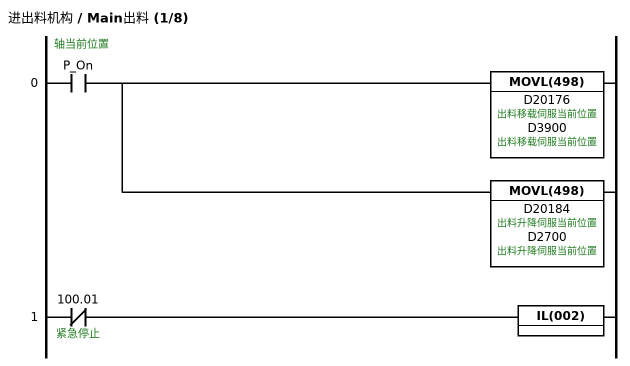
; [picture p48: 进出料机构 / Main出料, rungs 0-1]
; rung 0: 轴当前位置
LD P_On
MOVL(498) D20176 D3900  ; 出料移载伺服当前位置
MOVL(498) D20184 D2700  ; 出料升降伺服当前位置
; rung 1
LDNOT 100.01  ; 紧急停止
IL(002)

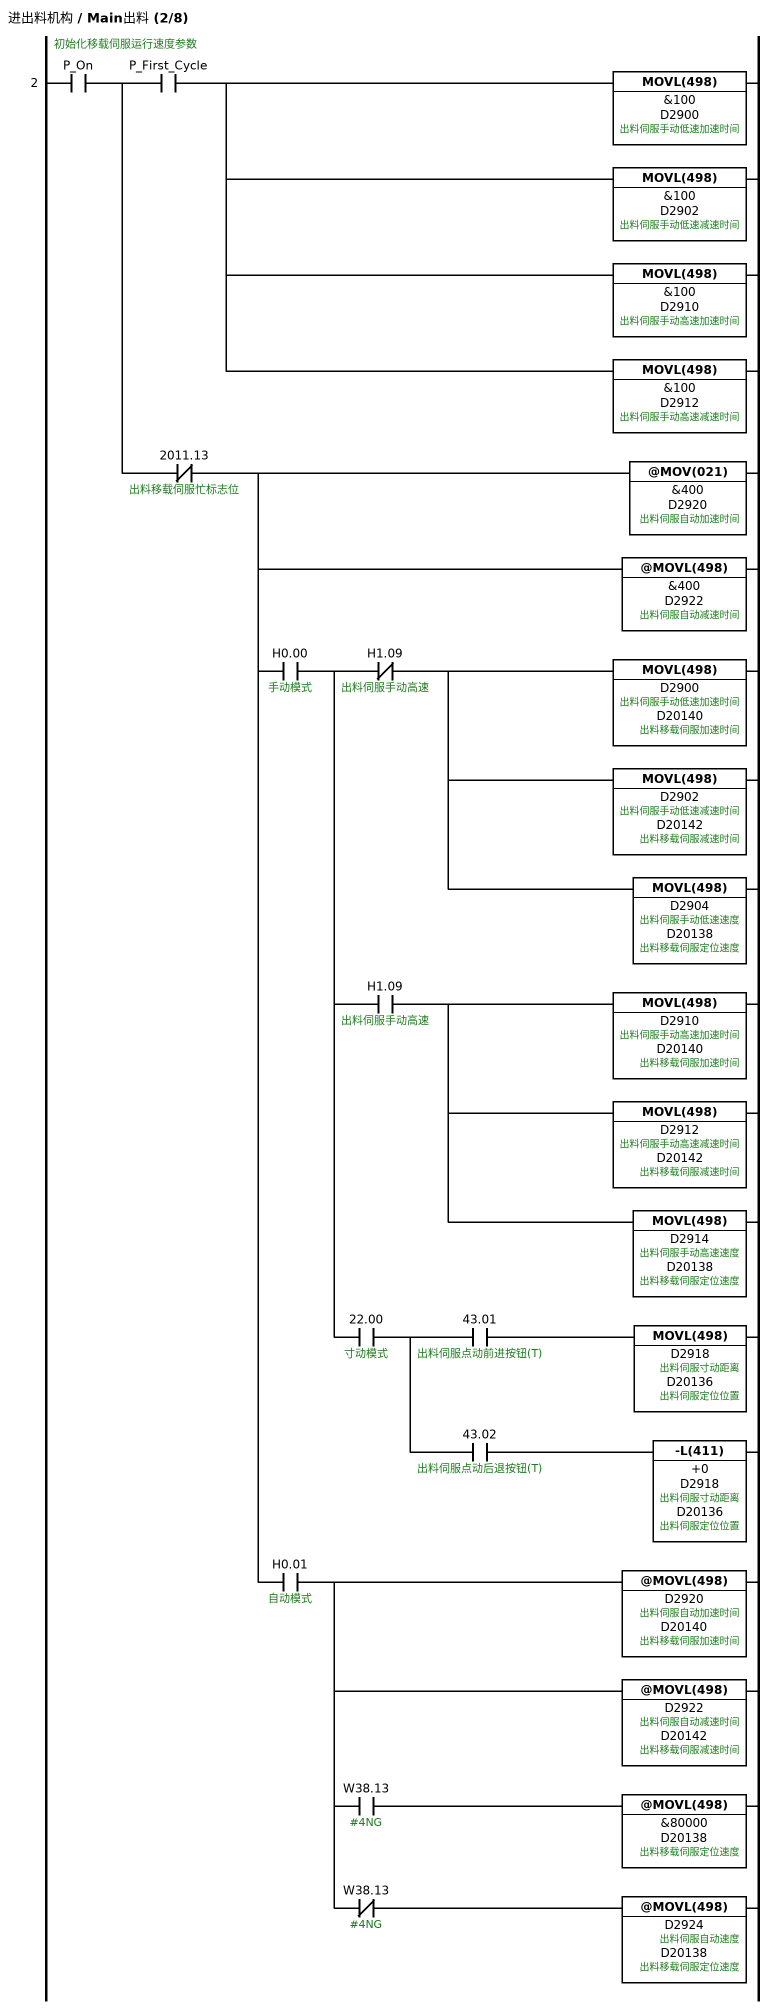
; rung 2: 初始化移载伺服运行速度参数
LD P_On
OUT TR0
AND P_First_Cycle
MOVL(498) &100 D2900  ; 出料伺服手动低速加速时间
MOVL(498) &100 D2902  ; 出料伺服手动低速减速时间
MOVL(498) &100 D2910  ; 出料伺服手动高速加速时间
MOVL(498) &100 D2912  ; 出料伺服手动高速减速时间
LD TR0
ANDNOT 2011.13  ; 出料移载伺服忙标志位
OUT TR0
@MOV(021) &400 D2920  ; 出料伺服自动加速时间
@MOVL(498) &400 D2922  ; 出料伺服自动减速时间
AND H0.00  ; 手动模式
OUT TR1
ANDNOT H1.09  ; 出料伺服手动高速
MOVL(498) D2900 D20140  ; 出料伺服手动低速加速时间, 出料移载伺服加速时间
MOVL(498) D2902 D20142  ; 出料伺服手动低速减速时间, 出料移载伺服减速时间
MOVL(498) D2904 D20138  ; 出料伺服手动低速速度, 出料移载伺服定位速度
LD TR1
AND H1.09  ; 出料伺服手动高速
MOVL(498) D2910 D20140  ; 出料伺服手动高速加速时间, 出料移载伺服加速时间
MOVL(498) D2912 D20142  ; 出料伺服手动高速减速时间, 出料移载伺服减速时间
MOVL(498) D2914 D20138  ; 出料伺服手动高速速度, 出料移载伺服定位速度
LD TR1
AND 22.00  ; 寸动模式
OUT TR1
AND 43.01  ; 出料伺服点动前进按钮(T)
MOVL(498) D2918 D20136  ; 出料伺服寸动距离, 出料伺服定位位置
LD TR1
AND 43.02  ; 出料伺服点动后退按钮(T)
-L(411) +0 D2918 D20136  ; 出料伺服寸动距离, 出料伺服定位位置
LD TR0
AND H0.01  ; 自动模式
OUT TR0
@MOVL(498) D2920 D20140  ; 出料伺服自动加速时间, 出料移载伺服加速时间
@MOVL(498) D2922 D20142  ; 出料伺服自动减速时间, 出料移载伺服减速时间
AND W38.13  ; #4NG
@MOVL(498) &80000 D20138  ; 出料移载伺服定位速度
LD TR0
ANDNOT W38.13  ; #4NG
@MOVL(498) D2924 D20138  ; 出料伺服自动速度, 出料移载伺服定位速度

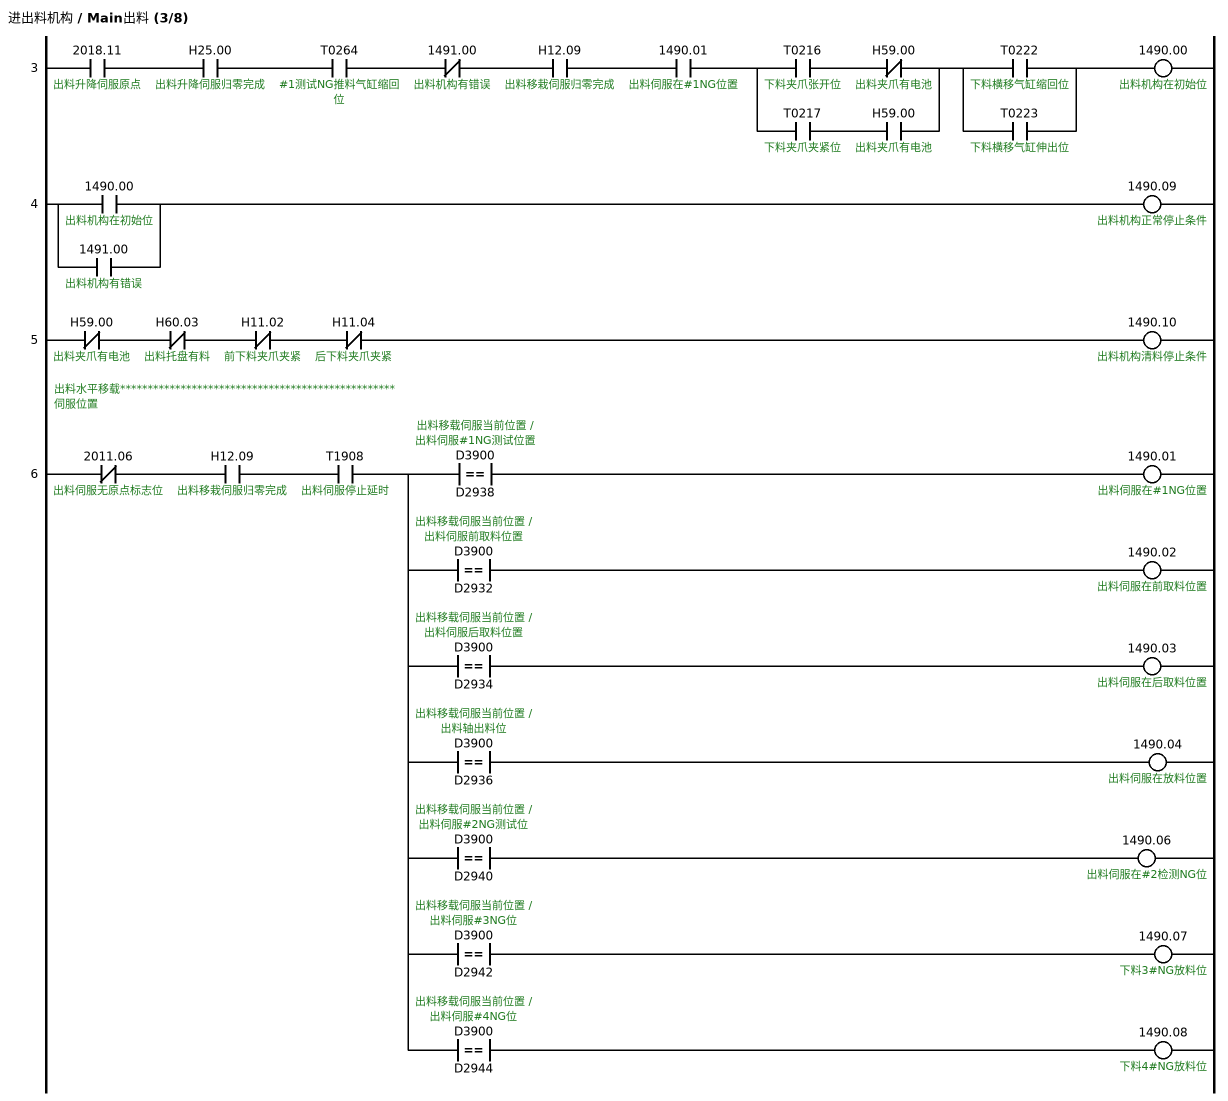
; rung 3
LD 2018.11  ; 出料升降伺服原点
AND H25.00  ; 出料升降伺服归零完成
AND T0264  ; #1测试NG推料气缸缩回位
ANDNOT 1491.00  ; 出料机构有错误
AND H12.09  ; 出料移栽伺服归零完成
AND 1490.01  ; 出料伺服在#1NG位置
LD T0216  ; 下料夹爪张开位
ANDNOT H59.00  ; 出料夹爪有电池
LD T0217  ; 下料夹爪夹紧位
AND H59.00  ; 出料夹爪有电池
ORLD
ANDLD
LD T0222  ; 下料横移气缸缩回位
OR T0223  ; 下料横移气缸伸出位
ANDLD
OUT 1490.00  ; 出料机构在初始位
; rung 4
LD 1490.00  ; 出料机构在初始位
OR 1491.00  ; 出料机构有错误
OUT 1490.09  ; 出料机构正常停止条件
; rung 5
LDNOT H59.00  ; 出料夹爪有电池
ANDNOT H60.03  ; 出料托盘有料
ANDNOT H11.02  ; 前下料夹爪夹紧
ANDNOT H11.04  ; 后下料夹爪夹紧
OUT 1490.10  ; 出料机构清料停止条件
; rung 6: 出料水平移载************************************************** / 伺服位置
LDNOT 2011.06  ; 出料伺服无原点标志位
AND H12.09  ; 出料移栽伺服归零完成
AND T1908  ; 出料伺服停止延时
OUT TR0
AND=SL(303) D3900 D2938  ; 出料移载伺服当前位置, 出料伺服#1NG测试位置
OUT 1490.01  ; 出料伺服在#1NG位置
LD TR0
AND=SL(303) D3900 D2932  ; 出料移载伺服当前位置, 出料伺服前取料位置
OUT 1490.02  ; 出料伺服在前取料位置
LD TR0
AND=SL(303) D3900 D2934  ; 出料移载伺服当前位置, 出料伺服后取料位置
OUT 1490.03  ; 出料伺服在后取料位置
LD TR0
AND=SL(303) D3900 D2936  ; 出料移载伺服当前位置, 出料轴出料位
OUT 1490.04  ; 出料伺服在放料位置
LD TR0
AND=SL(303) D3900 D2940  ; 出料移载伺服当前位置, 出料伺服#2NG测试位
OUT 1490.06  ; 出料伺服在#2检测NG位
LD TR0
AND=SL(303) D3900 D2942  ; 出料移载伺服当前位置, 出料伺服#3NG位
OUT 1490.07  ; 下料3#NG放料位
LD TR0
AND=SL(303) D3900 D2944  ; 出料移载伺服当前位置, 出料伺服#4NG位
OUT 1490.08  ; 下料4#NG放料位

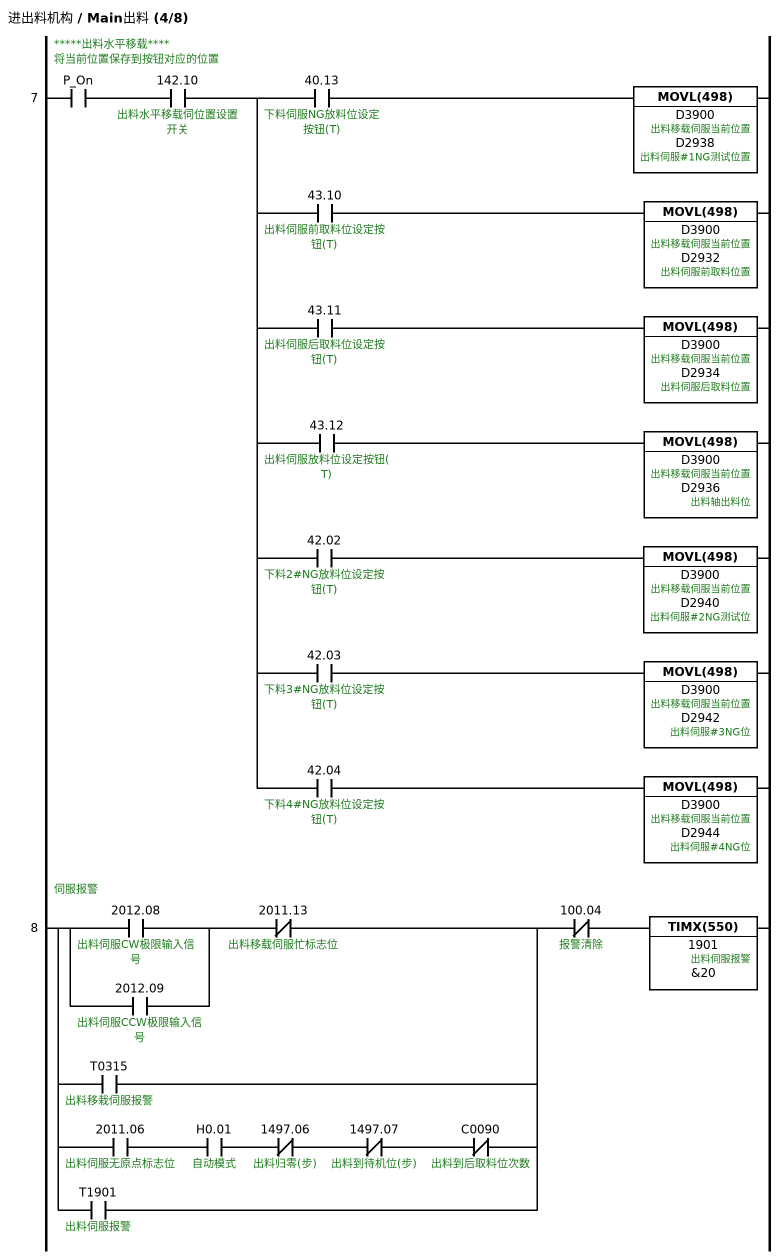
; rung 7: *****出料水平移载**** / 将当前位置保存到按钮对应的位置
LD P_On
AND 142.10  ; 出料水平移载伺位置设置开关
OUT TR0
AND 40.13  ; 下料伺服NG放料位设定按钮(T)
MOVL(498) D3900 D2938  ; 出料移载伺服当前位置, 出料伺服#1NG测试位置
LD TR0
AND 43.10  ; 出料伺服前取料位设定按钮(T)
MOVL(498) D3900 D2932  ; 出料移载伺服当前位置, 出料伺服前取料位置
LD TR0
AND 43.11  ; 出料伺服后取料位设定按钮(T)
MOVL(498) D3900 D2934  ; 出料移载伺服当前位置, 出料伺服后取料位置
LD TR0
AND 43.12  ; 出料伺服放料位设定按钮(T)
MOVL(498) D3900 D2936  ; 出料移载伺服当前位置, 出料轴出料位
LD TR0
AND 42.02  ; 下料2#NG放料位设定按钮(T)
MOVL(498) D3900 D2940  ; 出料移载伺服当前位置, 出料伺服#2NG测试位
LD TR0
AND 42.03  ; 下料3#NG放料位设定按钮(T)
MOVL(498) D3900 D2942  ; 出料移载伺服当前位置, 出料伺服#3NG位
LD TR0
AND 42.04  ; 下料4#NG放料位设定按钮(T)
MOVL(498) D3900 D2944  ; 出料移载伺服当前位置, 出料伺服#4NG位
; rung 8: 伺服报警
LD 2012.08  ; 出料伺服CW极限输入信号
OR 2012.09  ; 出料伺服CCW极限输入信号
ANDNOT 2011.13  ; 出料移载伺服忙标志位
OR T0315  ; 出料移栽伺服报警
LD 2011.06  ; 出料伺服无原点标志位
AND H0.01  ; 自动模式
ANDNOT 1497.06  ; 出料归零(步)
ANDNOT 1497.07  ; 出料到待机位(步)
ANDNOT C0090  ; 出料到后取料位次数
ORLD
OR T1901  ; 出料伺服报警
ANDNOT 100.04  ; 报警清除
TIMX(550) 1901 &20  ; 出料伺服报警

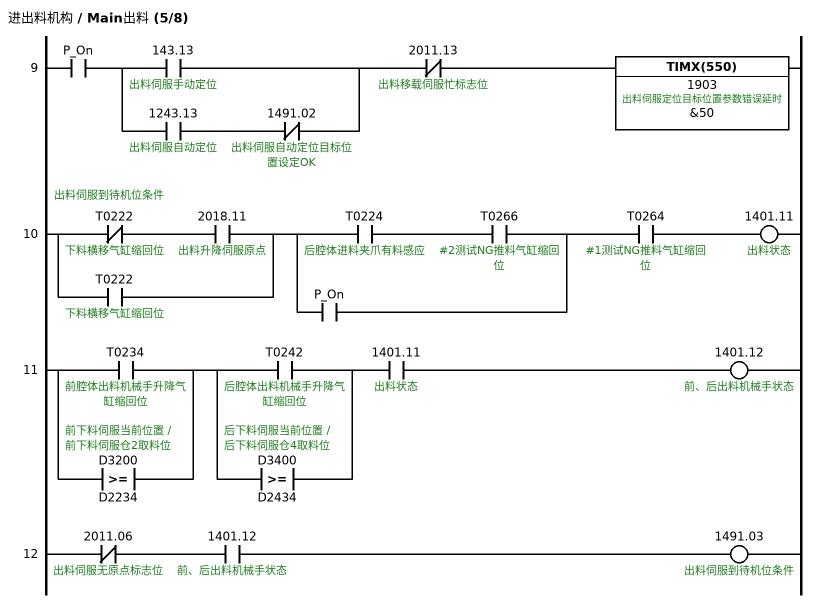
; rung 9
LD P_On
LD 143.13  ; 出料伺服手动定位
LD 1243.13  ; 出料伺服自动定位
ANDNOT 1491.02  ; 出料伺服自动定位目标位置设定OK
ORLD
ANDLD
ANDNOT 2011.13  ; 出料移载伺服忙标志位
TIMX(550) 1903 &50  ; 出料伺服定位目标位置参数错误延时
; rung 10: 出料伺服到待机位条件
LDNOT T0222  ; 下料横移气缸缩回位
AND 2018.11  ; 出料升降伺服原点
OR T0222  ; 下料横移气缸缩回位
LD T0224  ; 后腔体进料夹爪有料感应
AND T0266  ; #2测试NG推料气缸缩回位
OR P_On
ANDLD
AND T0264  ; #1测试NG推料气缸缩回位
OUT 1401.11  ; 出料状态
; rung 11
LD T0234  ; 前腔体出料机械手升降气缸缩回位
OR>=SL(328) D3200 D2234  ; 前下料伺服当前位置, 前下料伺服仓2取料位
LD T0242  ; 后腔体出料机械手升降气缸缩回位
OR>=SL(328) D3400 D2434  ; 后下料伺服当前位置, 后下料伺服仓4取料位
ANDLD
AND 1401.11  ; 出料状态
OUT 1401.12  ; 前、后出料机械手状态
; rung 12
LDNOT 2011.06  ; 出料伺服无原点标志位
AND 1401.12  ; 前、后出料机械手状态
OUT 1491.03  ; 出料伺服到待机位条件

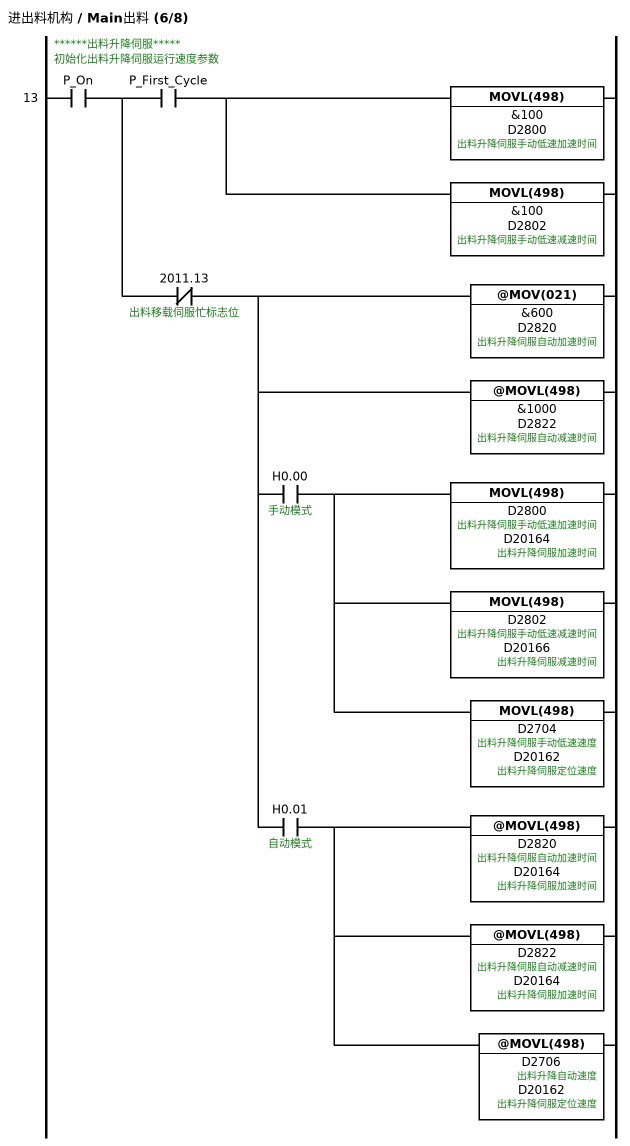
; rung 13: ******出料升降伺服***** / 初始化出料升降伺服运行速度参数
LD P_On
OUT TR0
AND P_First_Cycle
MOVL(498) &100 D2800  ; 出料升降伺服手动低速加速时间
MOVL(498) &100 D2802  ; 出料升降伺服手动低速减速时间
LD TR0
ANDNOT 2011.13  ; 出料移载伺服忙标志位
OUT TR0
@MOV(021) &600 D2820  ; 出料升降伺服自动加速时间
@MOVL(498) &1000 D2822  ; 出料升降伺服自动减速时间
AND H0.00  ; 手动模式
MOVL(498) D2800 D20164  ; 出料升降伺服手动低速加速时间, 出料升降伺服加速时间
MOVL(498) D2802 D20166  ; 出料升降伺服手动低速减速时间, 出料升降伺服减速时间
MOVL(498) D2704 D20162  ; 出料升降伺服手动低速速度, 出料升降伺服定位速度
LD TR0
AND H0.01  ; 自动模式
@MOVL(498) D2820 D20164  ; 出料升降伺服自动加速时间, 出料升降伺服加速时间
@MOVL(498) D2822 D20164  ; 出料升降伺服自动减速时间, 出料升降伺服加速时间
@MOVL(498) D2706 D20162  ; 出料升降自动速度, 出料升降伺服定位速度

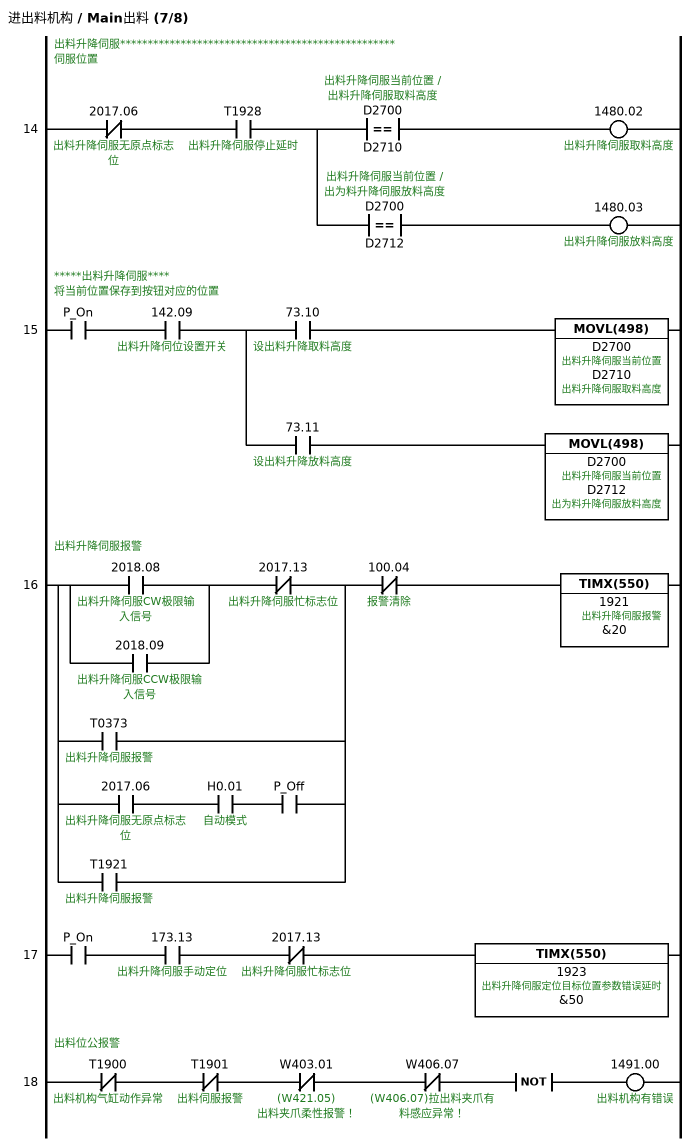
; rung 14: 出料升降伺服************************************************** / 伺服位置
LDNOT 2017.06  ; 出料升降伺服无原点标志位
AND T1928  ; 出料升降伺服停止延时
OUT TR0
AND=SL(303) D2700 D2710  ; 出料升降伺服当前位置, 出料升降伺服取料高度
OUT 1480.02  ; 出料升降伺服取料高度
LD TR0
AND=SL(303) D2700 D2712  ; 出料升降伺服当前位置, 出为料升降伺服放料高度
OUT 1480.03  ; 出料升降伺服放料高度
; rung 15: *****出料升降伺服**** / 将当前位置保存到按钮对应的位置
LD P_On
AND 142.09  ; 出料升降伺位设置开关
OUT TR0
AND 73.10  ; 设出料升降取料高度
MOVL(498) D2700 D2710  ; 出料升降伺服当前位置, 出料升降伺服取料高度
LD TR0
AND 73.11  ; 设出料升降放料高度
MOVL(498) D2700 D2712  ; 出料升降伺服当前位置, 出为料升降伺服放料高度
; rung 16: 出料升降伺服报警
LD 2018.08  ; 出料升降伺服CW极限输入信号
OR 2018.09  ; 出料升降伺服CCW极限输入信号
ANDNOT 2017.13  ; 出料升降伺服忙标志位
OR T0373  ; 出料升降伺服报警
LD 2017.06  ; 出料升降伺服无原点标志位
AND H0.01  ; 自动模式
AND P_Off
ORLD
OR T1921  ; 出料升降伺服报警
ANDNOT 100.04  ; 报警清除
TIMX(550) 1921 &20  ; 出料升降伺服报警
; rung 17
LD P_On
AND 173.13  ; 出料升降伺服手动定位
ANDNOT 2017.13  ; 出料升降伺服忙标志位
TIMX(550) 1923 &50  ; 出料升降伺服定位目标位置参数错误延时
; rung 18: 出料位公报警
LDNOT T1900  ; 出料机构气缸动作异常
ANDNOT T1901  ; 出料伺服报警
ANDNOT W403.01  ; (W421.05) 出料夹爪柔性报警！
ANDNOT W406.07  ; (W406.07)拉出料夹爪有料感应异常！
NOT(520)
OUT 1491.00  ; 出料机构有错误

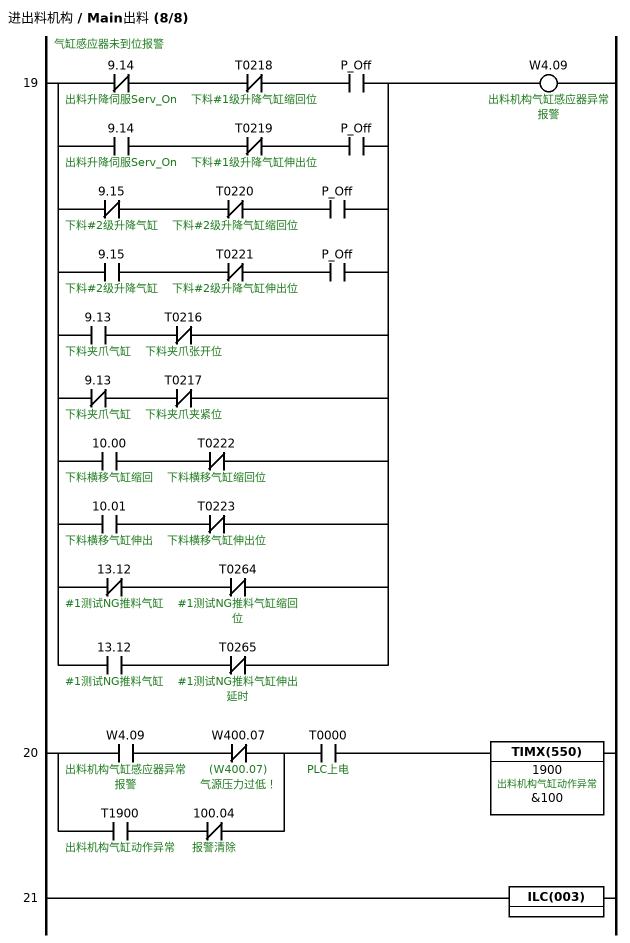
; rung 19: 气缸感应器未到位报警
LDNOT 9.14  ; 出料升降伺服Serv_On
ANDNOT T0218  ; 下料#1级升降气缸缩回位
AND P_Off
LD 9.14  ; 出料升降伺服Serv_On
ANDNOT T0219  ; 下料#1级升降气缸伸出位
AND P_Off
ORLD
LDNOT 9.15  ; 下料#2级升降气缸
ANDNOT T0220  ; 下料#2级升降气缸缩回位
AND P_Off
ORLD
LD 9.15  ; 下料#2级升降气缸
ANDNOT T0221  ; 下料#2级升降气缸伸出位
AND P_Off
ORLD
LD 9.13  ; 下料夹爪气缸
ANDNOT T0216  ; 下料夹爪张开位
ORLD
LDNOT 9.13  ; 下料夹爪气缸
ANDNOT T0217  ; 下料夹爪夹紧位
ORLD
LD 10.00  ; 下料横移气缸缩回
ANDNOT T0222  ; 下料横移气缸缩回位
ORLD
LD 10.01  ; 下料横移气缸伸出
ANDNOT T0223  ; 下料横移气缸伸出位
ORLD
LDNOT 13.12  ; #1测试NG推料气缸
ANDNOT T0264  ; #1测试NG推料气缸缩回位
ORLD
LD 13.12  ; #1测试NG推料气缸
ANDNOT T0265  ; #1测试NG推料气缸伸出延时
ORLD
OUT W4.09  ; 出料机构气缸感应器异常报警
; rung 20
LD W4.09  ; 出料机构气缸感应器异常报警
ANDNOT W400.07  ; (W400.07) 气源压力过低！
LD T1900  ; 出料机构气缸动作异常
ANDNOT 100.04  ; 报警清除
ORLD
AND T0000  ; PLC上电
TIMX(550) 1900 &100  ; 出料机构气缸动作异常
; rung 21
ILC(003)

### Section 工站复位

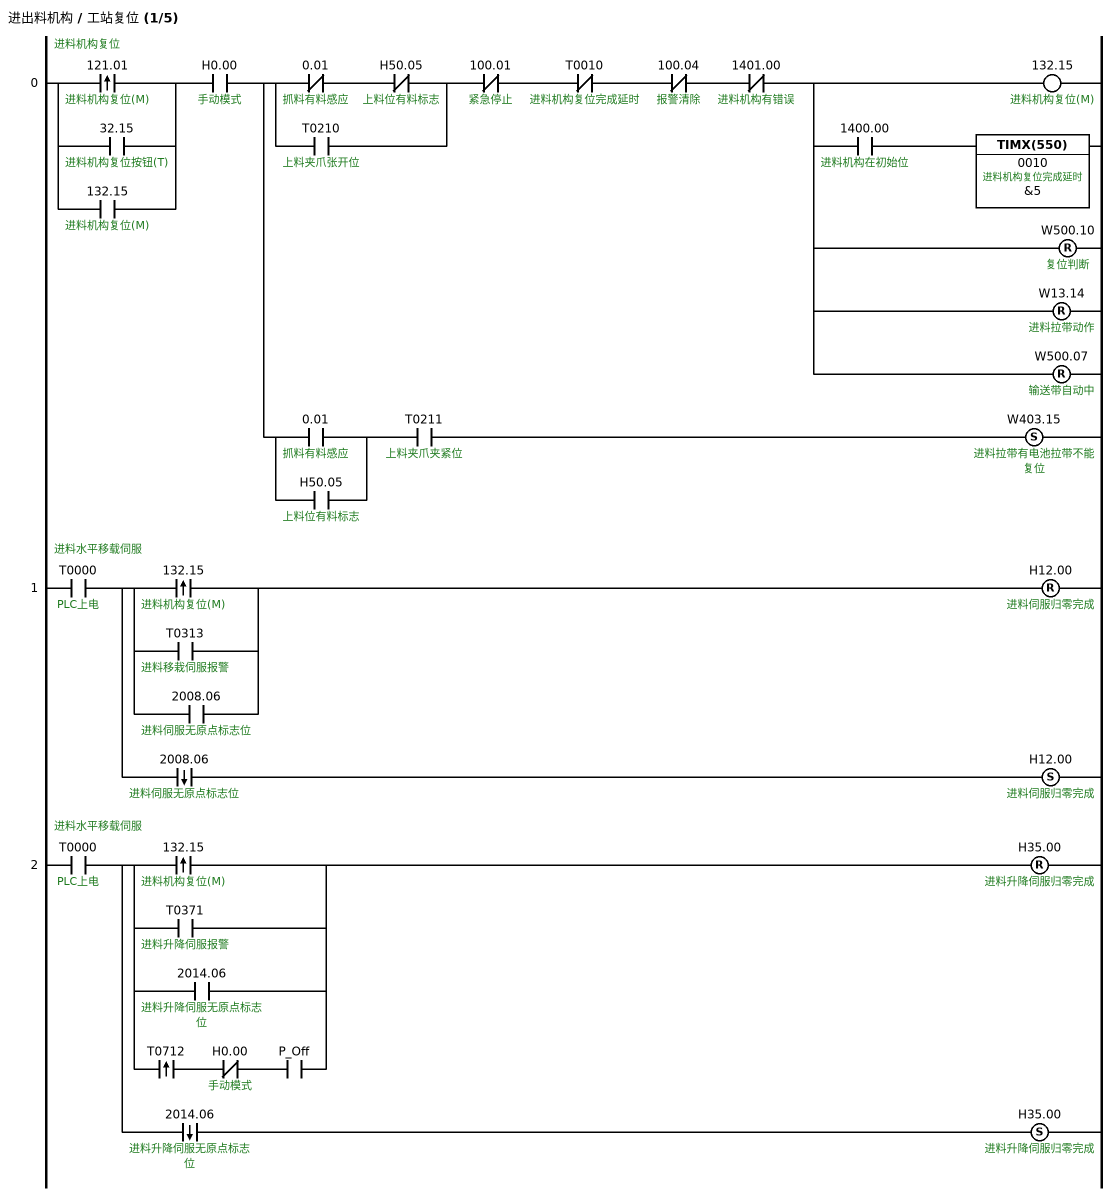
; rung 0: 进料机构复位
@LD 121.01  ; 进料机构复位(M)
OR 32.15  ; 进料机构复位按钮(T)
OR 132.15  ; 进料机构复位(M)
AND H0.00  ; 手动模式
OUT TR0
LDNOT 0.01  ; 抓料有料感应
ANDNOT H50.05  ; 上料位有料标志
OR T0210  ; 上料夹爪张开位
ANDLD
ANDNOT 100.01  ; 紧急停止
ANDNOT T0010  ; 进料机构复位完成延时
ANDNOT 100.04  ; 报警清除
ANDNOT 1401.00  ; 进料机构有错误
OUT TR1
OUT 132.15  ; 进料机构复位(M)
AND 1400.00  ; 进料机构在初始位
TIMX(550) 0010 &5  ; 进料机构复位完成延时
LD TR1
RSET W500.10  ; 复位判断
RSET W13.14  ; 进料拉带动作
RSET W500.07  ; 输送带自动中
LD TR0
LD 0.01  ; 抓料有料感应
OR H50.05  ; 上料位有料标志
ANDLD
AND T0211  ; 上料夹爪夹紧位
SET W403.15  ; 进料拉带有电池拉带不能复位
; rung 1: 进料水平移载伺服
LD T0000  ; PLC上电
OUT TR0
@LD 132.15  ; 进料机构复位(M)
OR T0313  ; 进料移栽伺服报警
OR 2008.06  ; 进料伺服无原点标志位
ANDLD
RSET H12.00  ; 进料伺服归零完成
LD TR0
%AND 2008.06  ; 进料伺服无原点标志位
SET H12.00  ; 进料伺服归零完成
; rung 2: 进料水平移载伺服
LD T0000  ; PLC上电
OUT TR0
@LD 132.15  ; 进料机构复位(M)
OR T0371  ; 进料升降伺服报警
OR 2014.06  ; 进料升降伺服无原点标志位
@LD T0712
ANDNOT H0.00  ; 手动模式
AND P_Off
ORLD
ANDLD
RSET H35.00  ; 进料升降伺服归零完成
LD TR0
%AND 2014.06  ; 进料升降伺服无原点标志位
SET H35.00  ; 进料升降伺服归零完成

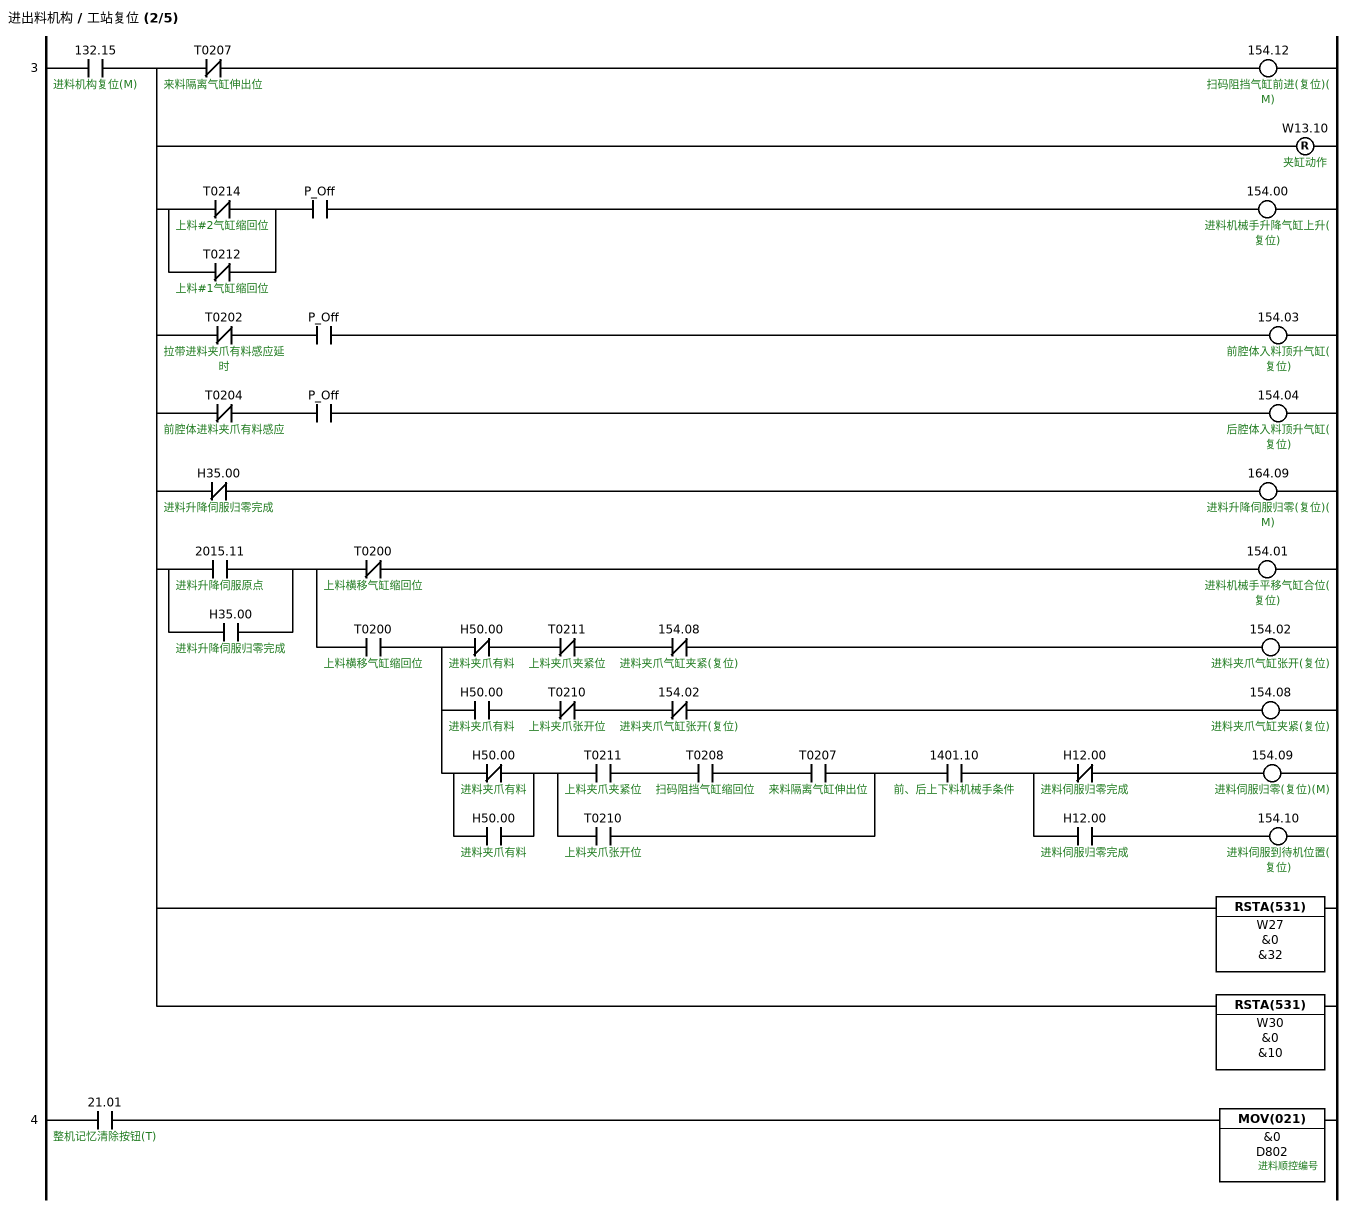
; rung 3
LD 132.15  ; 进料机构复位(M)
OUT TR0
ANDNOT T0207  ; 来料隔离气缸伸出位
OUT 154.12  ; 扫码阻挡气缸前进(复位)(M)
LD TR0
RSET W13.10  ; 夹缸动作
LDNOT T0214  ; 上料#2气缸缩回位
ORNOT T0212  ; 上料#1气缸缩回位
ANDLD
AND P_Off
OUT 154.00  ; 进料机械手升降气缸上升(复位)
LD TR0
ANDNOT T0202  ; 拉带进料夹爪有料感应延时
AND P_Off
OUT 154.03  ; 前腔体入料顶升气缸(复位)
LD TR0
ANDNOT T0204  ; 前腔体进料夹爪有料感应
AND P_Off
OUT 154.04  ; 后腔体入料顶升气缸(复位)
LD TR0
ANDNOT H35.00  ; 进料升降伺服归零完成
OUT 164.09  ; 进料升降伺服归零(复位)(M)
LD TR0
LD 2015.11  ; 进料升降伺服原点
OR H35.00  ; 进料升降伺服归零完成
ANDLD
OUT TR1
ANDNOT T0200  ; 上料横移气缸缩回位
OUT 154.01  ; 进料机械手平移气缸合位(复位)
LD TR1
AND T0200  ; 上料横移气缸缩回位
OUT TR1
ANDNOT H50.00  ; 进料夹爪有料
ANDNOT T0211  ; 上料夹爪夹紧位
ANDNOT 154.08  ; 进料夹爪气缸夹紧(复位)
OUT 154.02  ; 进料夹爪气缸张开(复位)
LD TR1
AND H50.00  ; 进料夹爪有料
ANDNOT T0210  ; 上料夹爪张开位
ANDNOT 154.02  ; 进料夹爪气缸张开(复位)
OUT 154.08  ; 进料夹爪气缸夹紧(复位)
LD TR1
LDNOT H50.00  ; 进料夹爪有料
OR H50.00  ; 进料夹爪有料
ANDLD
LD T0211  ; 上料夹爪夹紧位
AND T0208  ; 扫码阻挡气缸缩回位
AND T0207  ; 来料隔离气缸伸出位
OR T0210  ; 上料夹爪张开位
ANDLD
AND 1401.10  ; 前、后上下料机械手条件
OUT TR1
ANDNOT H12.00  ; 进料伺服归零完成
OUT 154.09  ; 进料伺服归零(复位)(M)
LD TR1
AND H12.00  ; 进料伺服归零完成
OUT 154.10  ; 进料伺服到待机位置(复位)
LD TR0
RSTA(531) W27 &0 &32
RSTA(531) W30 &0 &10
; rung 4
LD 21.01  ; 整机记忆清除按钮(T)
MOV(021) &0 D802  ; 进料顺控编号

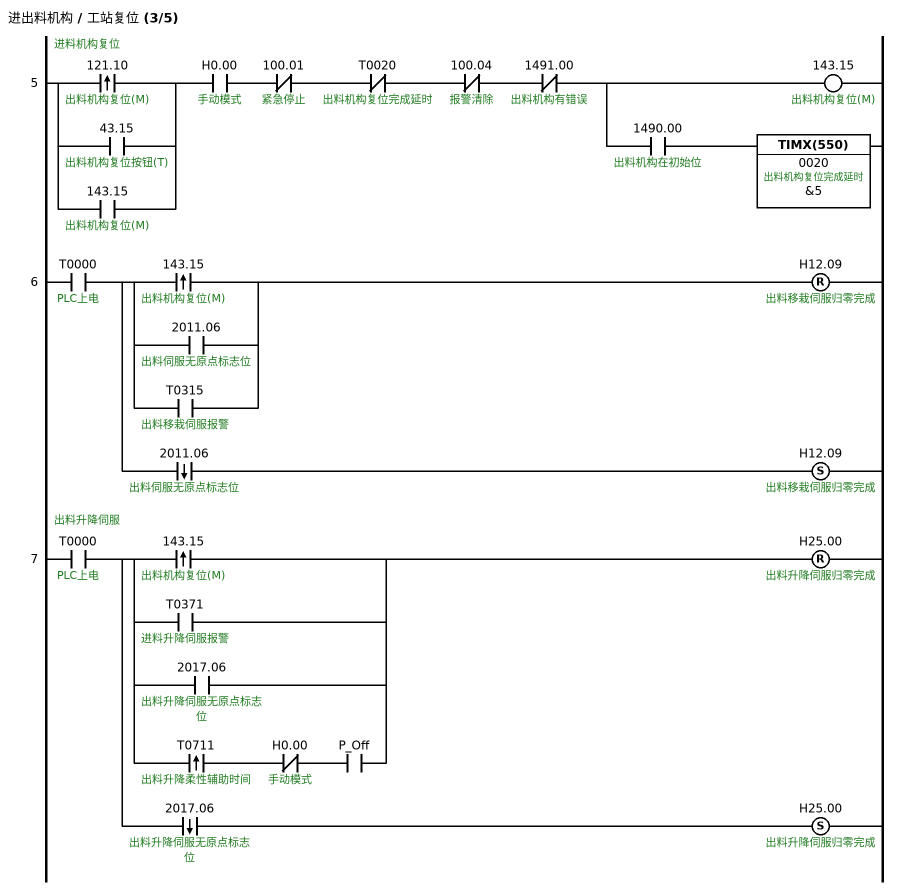
; rung 5: 进料机构复位
@LD 121.10  ; 出料机构复位(M)
OR 43.15  ; 出料机构复位按钮(T)
OR 143.15  ; 出料机构复位(M)
AND H0.00  ; 手动模式
ANDNOT 100.01  ; 紧急停止
ANDNOT T0020  ; 出料机构复位完成延时
ANDNOT 100.04  ; 报警清除
ANDNOT 1491.00  ; 出料机构有错误
OUT 143.15  ; 出料机构复位(M)
AND 1490.00  ; 出料机构在初始位
TIMX(550) 0020 &5  ; 出料机构复位完成延时
; rung 6
LD T0000  ; PLC上电
OUT TR0
@LD 143.15  ; 出料机构复位(M)
OR 2011.06  ; 出料伺服无原点标志位
OR T0315  ; 出料移栽伺服报警
ANDLD
RSET H12.09  ; 出料移栽伺服归零完成
LD TR0
%AND 2011.06  ; 出料伺服无原点标志位
SET H12.09  ; 出料移栽伺服归零完成
; rung 7: 出料升降伺服
LD T0000  ; PLC上电
OUT TR0
@LD 143.15  ; 出料机构复位(M)
OR T0371  ; 进料升降伺服报警
OR 2017.06  ; 出料升降伺服无原点标志位
@LD T0711  ; 出料升降柔性辅助时间
ANDNOT H0.00  ; 手动模式
AND P_Off
ORLD
ANDLD
RSET H25.00  ; 出料升降伺服归零完成
LD TR0
%AND 2017.06  ; 出料升降伺服无原点标志位
SET H25.00  ; 出料升降伺服归零完成

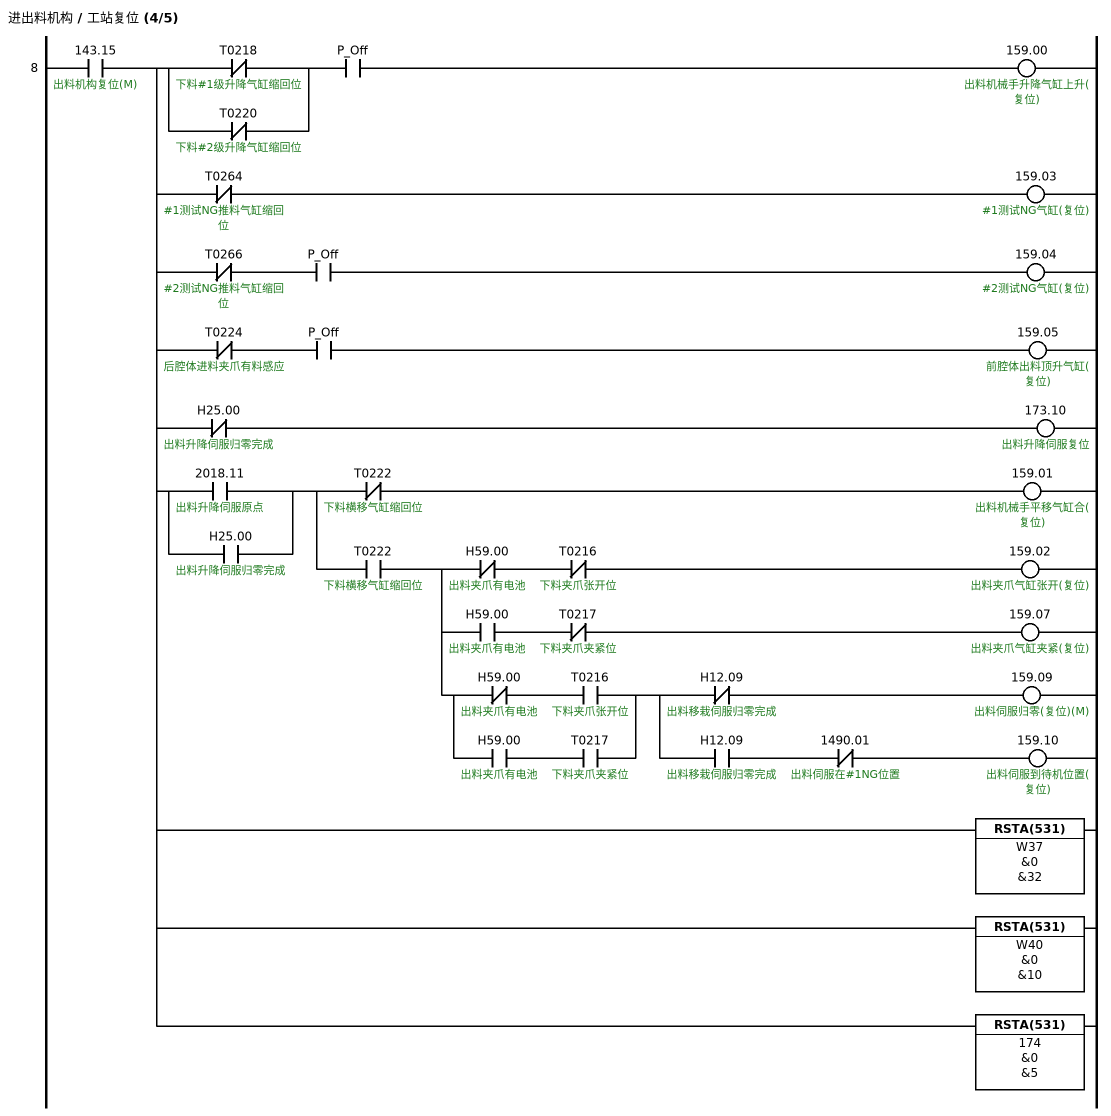
; rung 8
LD 143.15  ; 出料机构复位(M)
OUT TR0
LDNOT T0218  ; 下料#1级升降气缸缩回位
ORNOT T0220  ; 下料#2级升降气缸缩回位
ANDLD
AND P_Off
OUT 159.00  ; 出料机械手升降气缸上升(复位)
LD TR0
ANDNOT T0264  ; #1测试NG推料气缸缩回位
OUT 159.03  ; #1测试NG气缸(复位)
LD TR0
ANDNOT T0266  ; #2测试NG推料气缸缩回位
AND P_Off
OUT 159.04  ; #2测试NG气缸(复位)
LD TR0
ANDNOT T0224  ; 后腔体进料夹爪有料感应
AND P_Off
OUT 159.05  ; 前腔体出料顶升气缸(复位)
LD TR0
ANDNOT H25.00  ; 出料升降伺服归零完成
OUT 173.10  ; 出料升降伺服复位
LD TR0
LD 2018.11  ; 出料升降伺服原点
OR H25.00  ; 出料升降伺服归零完成
ANDLD
OUT TR1
ANDNOT T0222  ; 下料横移气缸缩回位
OUT 159.01  ; 出料机械手平移气缸合(复位)
LD TR1
AND T0222  ; 下料横移气缸缩回位
OUT TR1
ANDNOT H59.00  ; 出料夹爪有电池
ANDNOT T0216  ; 下料夹爪张开位
OUT 159.02  ; 出料夹爪气缸张开(复位)
LD TR1
AND H59.00  ; 出料夹爪有电池
ANDNOT T0217  ; 下料夹爪夹紧位
OUT 159.07  ; 出料夹爪气缸夹紧(复位)
LD TR1
LDNOT H59.00  ; 出料夹爪有电池
AND T0216  ; 下料夹爪张开位
LD H59.00  ; 出料夹爪有电池
AND T0217  ; 下料夹爪夹紧位
ORLD
ANDLD
OUT TR1
ANDNOT H12.09  ; 出料移栽伺服归零完成
OUT 159.09  ; 出料伺服归零(复位)(M)
LD TR1
AND H12.09  ; 出料移栽伺服归零完成
ANDNOT 1490.01  ; 出料伺服在#1NG位置
OUT 159.10  ; 出料伺服到待机位置(复位)
LD TR0
RSTA(531) W37 &0 &32
RSTA(531) W40 &0 &10
RSTA(531) 174 &0 &5

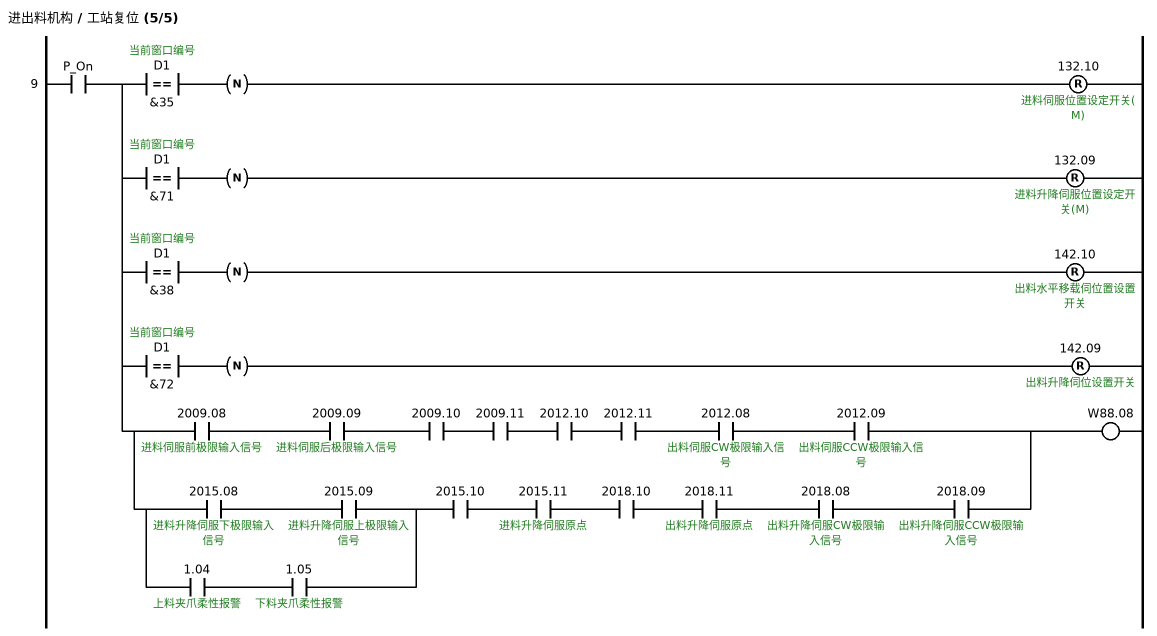
; rung 9
LD P_On
OUT TR0
AND=(300) D1 &35  ; 当前窗口编号
DOWN(522)
RSET 132.10  ; 进料伺服位置设定开关(M)
LD TR0
AND=(300) D1 &71  ; 当前窗口编号
DOWN(522)
RSET 132.09  ; 进料升降伺服位置设定开关(M)
LD TR0
AND=(300) D1 &38  ; 当前窗口编号
DOWN(522)
RSET 142.10  ; 出料水平移载伺位置设置开关
LD TR0
AND=(300) D1 &72  ; 当前窗口编号
DOWN(522)
RSET 142.09  ; 出料升降伺位设置开关
LD TR0
LD 2009.08  ; 进料伺服前极限输入信号
AND 2009.09  ; 进料伺服后极限输入信号
AND 2009.10
AND 2009.11
AND 2012.10
AND 2012.11
AND 2012.08  ; 出料伺服CW极限输入信号
AND 2012.09  ; 出料伺服CCW极限输入信号
LD 2015.08  ; 进料升降伺服下极限输入信号
AND 2015.09  ; 进料升降伺服上极限输入信号
LD 1.04  ; 上料夹爪柔性报警
AND 1.05  ; 下料夹爪柔性报警
ORLD
AND 2015.10
AND 2015.11  ; 进料升降伺服原点
AND 2018.10
AND 2018.11  ; 出料升降伺服原点
AND 2018.08  ; 出料升降伺服CW极限输入信号
AND 2018.09  ; 出料升降伺服CCW极限输入信号
ORLD
ANDLD
OUT W88.08

### Section 扫码

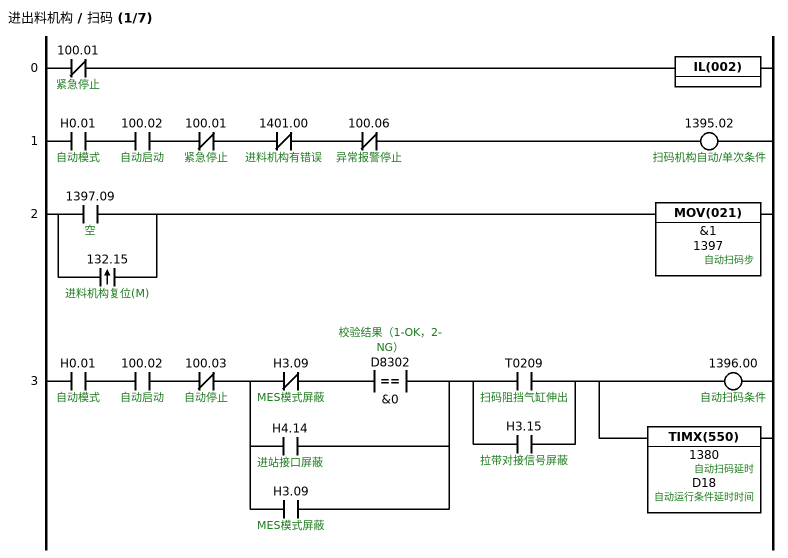
; rung 0
LDNOT 100.01  ; 紧急停止
IL(002)
; rung 1
LD H0.01  ; 自动模式
AND 100.02  ; 自动启动
ANDNOT 100.01  ; 紧急停止
ANDNOT 1401.00  ; 进料机构有错误
ANDNOT 100.06  ; 异常报警停止
OUT 1395.02  ; 扫码机构自动/单次条件
; rung 2
LD 1397.09  ; 空
@OR 132.15  ; 进料机构复位(M)
MOV(021) &1 1397  ; 自动扫码步
; rung 3
LD H0.01  ; 自动模式
AND 100.02  ; 自动启动
ANDNOT 100.03  ; 自动停止
LDNOT H3.09  ; MES模式屏蔽
AND=(300) D8302 &0  ; 校验结果（1-OK，2-NG）
OR H4.14  ; 进站接口屏蔽
OR H3.09  ; MES模式屏蔽
ANDLD
LD T0209  ; 扫码阻挡气缸伸出
OR H3.15  ; 拉带对接信号屏蔽
ANDLD
OUT 1396.00  ; 自动扫码条件
TIMX(550) 1380 D18  ; 自动运行条件延时时间, 自动扫码延时

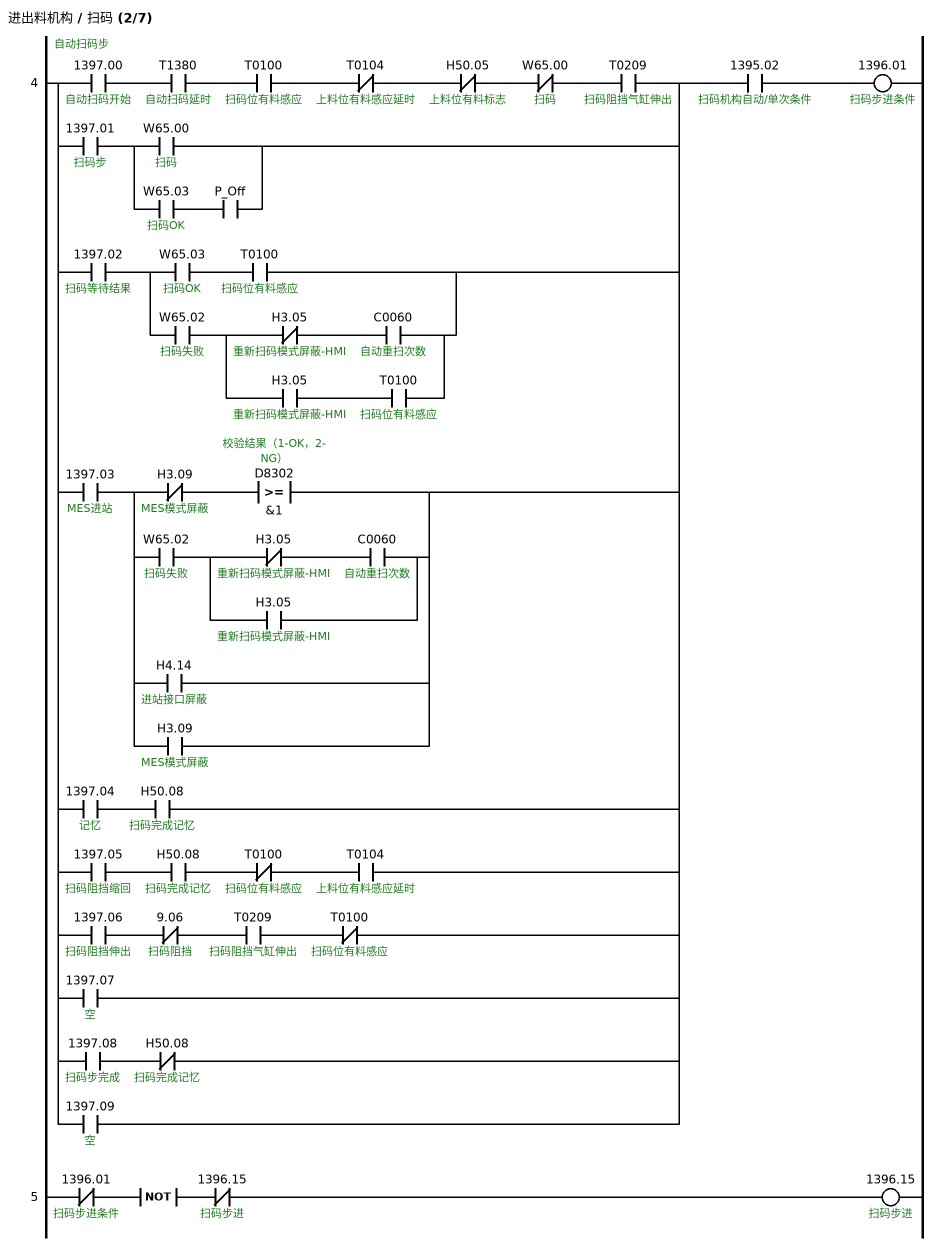
; rung 4: 自动扫码步
LD 1397.00  ; 自动扫码开始
AND T1380  ; 自动扫码延时
AND T0100  ; 扫码位有料感应
ANDNOT T0104  ; 上料位有料感应延时
ANDNOT H50.05  ; 上料位有料标志
ANDNOT W65.00  ; 扫码
AND T0209  ; 扫码阻挡气缸伸出
LD 1397.01  ; 扫码步
LD W65.00  ; 扫码
LD W65.03  ; 扫码OK
AND P_Off
ORLD
ANDLD
ORLD
LD 1397.02  ; 扫码等待结果
LD W65.03  ; 扫码OK
AND T0100  ; 扫码位有料感应
LD W65.02  ; 扫码失败
LDNOT H3.05  ; 重新扫码模式屏蔽-HMI
AND C0060  ; 自动重扫次数
LD H3.05  ; 重新扫码模式屏蔽-HMI
AND T0100  ; 扫码位有料感应
ORLD
ANDLD
ORLD
ANDLD
ORLD
LD 1397.03  ; MES进站
LDNOT H3.09  ; MES模式屏蔽
AND>=(325) D8302 &1  ; 校验结果（1-OK，2-NG）
LD W65.02  ; 扫码失败
LDNOT H3.05  ; 重新扫码模式屏蔽-HMI
AND C0060  ; 自动重扫次数
OR H3.05  ; 重新扫码模式屏蔽-HMI
ANDLD
ORLD
OR H4.14  ; 进站接口屏蔽
OR H3.09  ; MES模式屏蔽
ANDLD
ORLD
LD 1397.04  ; 记忆
AND H50.08  ; 扫码完成记忆
ORLD
LD 1397.05  ; 扫码阻挡缩回
AND H50.08  ; 扫码完成记忆
ANDNOT T0100  ; 扫码位有料感应
AND T0104  ; 上料位有料感应延时
ORLD
LD 1397.06  ; 扫码阻挡伸出
ANDNOT 9.06  ; 扫码阻挡
AND T0209  ; 扫码阻挡气缸伸出
ANDNOT T0100  ; 扫码位有料感应
ORLD
OR 1397.07  ; 空
LD 1397.08  ; 扫码步完成
ANDNOT H50.08  ; 扫码完成记忆
ORLD
OR 1397.09  ; 空
AND 1395.02  ; 扫码机构自动/单次条件
OUT 1396.01  ; 扫码步进条件
; rung 5
LDNOT 1396.01  ; 扫码步进条件
NOT(520)
ANDNOT 1396.15  ; 扫码步进
OUT 1396.15  ; 扫码步进

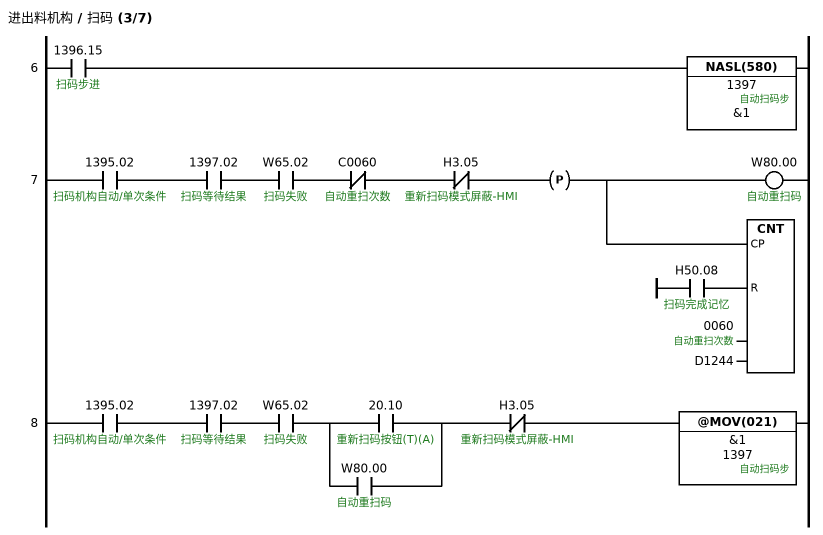
; rung 6
LD 1396.15  ; 扫码步进
NASL(580) 1397 &1  ; 自动扫码步
; rung 7
LD 1395.02  ; 扫码机构自动/单次条件
AND 1397.02  ; 扫码等待结果
AND W65.02  ; 扫码失败
ANDNOT C0060  ; 自动重扫次数
ANDNOT H3.05  ; 重新扫码模式屏蔽-HMI
UP(521)
OUT W80.00  ; 自动重扫码
LD H50.08  ; 扫码完成记忆
CNT 0060 D1244  ; 自动重扫次数
; rung 8
LD 1395.02  ; 扫码机构自动/单次条件
AND 1397.02  ; 扫码等待结果
AND W65.02  ; 扫码失败
LD 20.10  ; 重新扫码按钮(T)(A)
OR W80.00  ; 自动重扫码
ANDLD
ANDNOT H3.05  ; 重新扫码模式屏蔽-HMI
@MOV(021) &1 1397  ; 自动扫码步

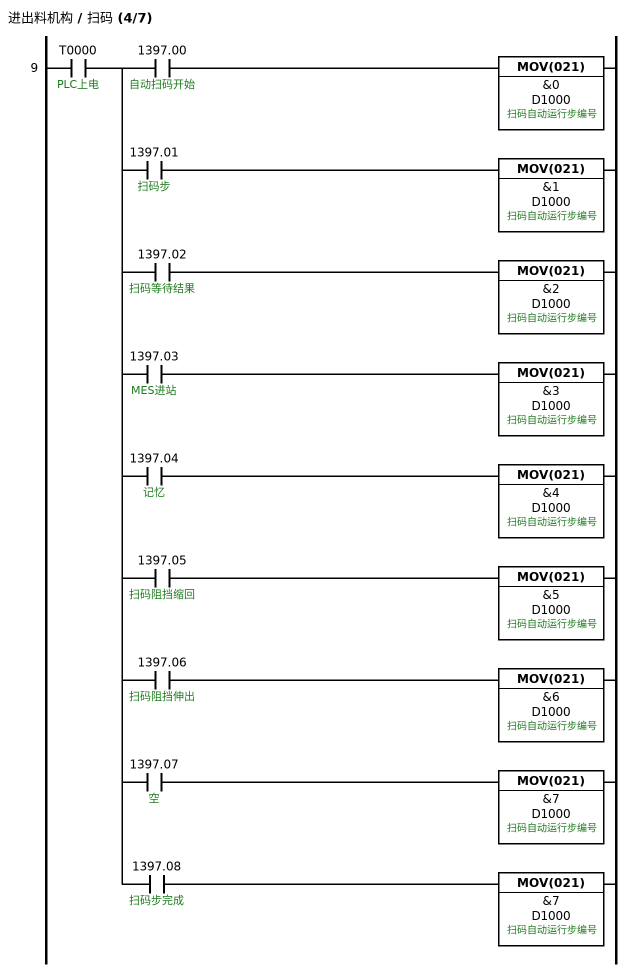
; rung 9
LD T0000  ; PLC上电
OUT TR0
AND 1397.00  ; 自动扫码开始
MOV(021) &0 D1000  ; 扫码自动运行步编号
LD TR0
AND 1397.01  ; 扫码步
MOV(021) &1 D1000  ; 扫码自动运行步编号
LD TR0
AND 1397.02  ; 扫码等待结果
MOV(021) &2 D1000  ; 扫码自动运行步编号
LD TR0
AND 1397.03  ; MES进站
MOV(021) &3 D1000  ; 扫码自动运行步编号
LD TR0
AND 1397.04  ; 记忆
MOV(021) &4 D1000  ; 扫码自动运行步编号
LD TR0
AND 1397.05  ; 扫码阻挡缩回
MOV(021) &5 D1000  ; 扫码自动运行步编号
LD TR0
AND 1397.06  ; 扫码阻挡伸出
MOV(021) &6 D1000  ; 扫码自动运行步编号
LD TR0
AND 1397.07  ; 空
MOV(021) &7 D1000  ; 扫码自动运行步编号
LD TR0
AND 1397.08  ; 扫码步完成
MOV(021) &7 D1000  ; 扫码自动运行步编号

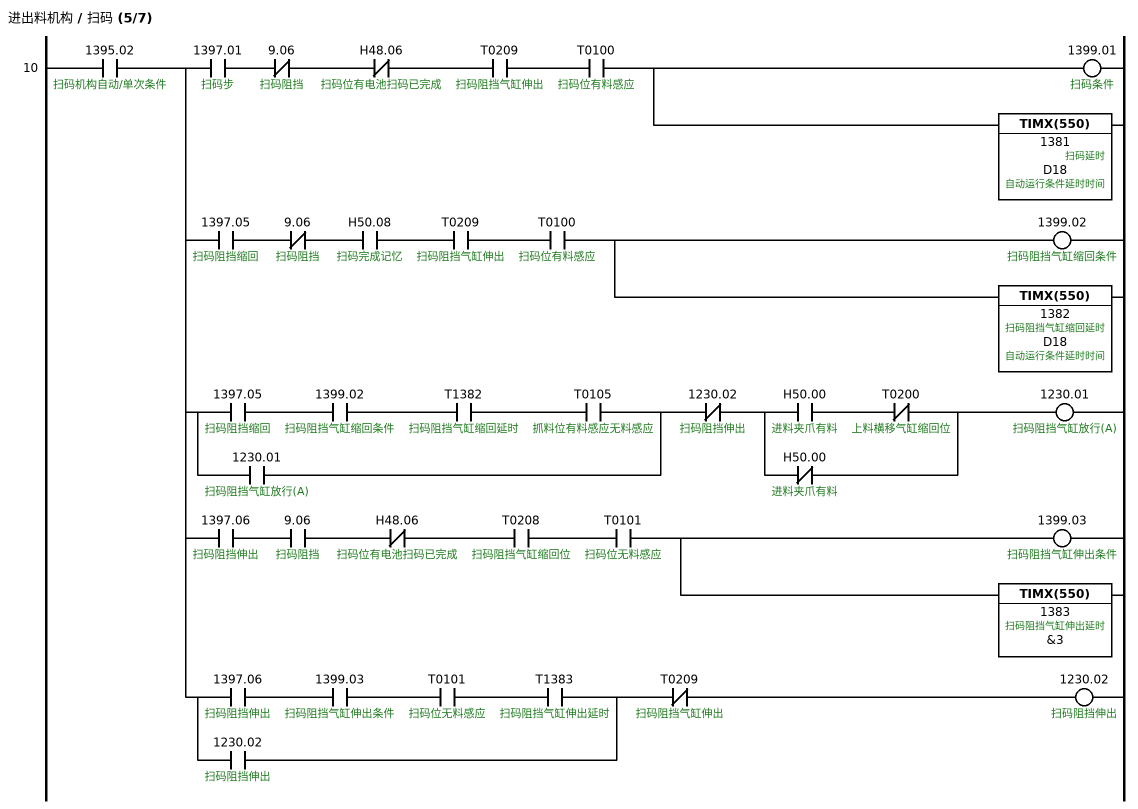
; rung 10
LD 1395.02  ; 扫码机构自动/单次条件
OUT TR0
AND 1397.01  ; 扫码步
ANDNOT 9.06  ; 扫码阻挡
ANDNOT H48.06  ; 扫码位有电池扫码已完成
AND T0209  ; 扫码阻挡气缸伸出
AND T0100  ; 扫码位有料感应
OUT 1399.01  ; 扫码条件
TIMX(550) 1381 D18  ; 自动运行条件延时时间, 扫码延时
LD TR0
AND 1397.05  ; 扫码阻挡缩回
ANDNOT 9.06  ; 扫码阻挡
AND H50.08  ; 扫码完成记忆
AND T0209  ; 扫码阻挡气缸伸出
AND T0100  ; 扫码位有料感应
OUT 1399.02  ; 扫码阻挡气缸缩回条件
TIMX(550) 1382 D18  ; 自动运行条件延时时间, 扫码阻挡气缸缩回延时
LD TR0
LD 1397.05  ; 扫码阻挡缩回
AND 1399.02  ; 扫码阻挡气缸缩回条件
AND T1382  ; 扫码阻挡气缸缩回延时
AND T0105  ; 抓料位有料感应无料感应
OR 1230.01  ; 扫码阻挡气缸放行(A)
ANDLD
ANDNOT 1230.02  ; 扫码阻挡伸出
LD H50.00  ; 进料夹爪有料
ANDNOT T0200  ; 上料横移气缸缩回位
ORNOT H50.00  ; 进料夹爪有料
ANDLD
OUT 1230.01  ; 扫码阻挡气缸放行(A)
LD TR0
AND 1397.06  ; 扫码阻挡伸出
AND 9.06  ; 扫码阻挡
ANDNOT H48.06  ; 扫码位有电池扫码已完成
AND T0208  ; 扫码阻挡气缸缩回位
AND T0101  ; 扫码位无料感应
OUT 1399.03  ; 扫码阻挡气缸伸出条件
TIMX(550) 1383 &3  ; 扫码阻挡气缸伸出延时
LD TR0
LD 1397.06  ; 扫码阻挡伸出
AND 1399.03  ; 扫码阻挡气缸伸出条件
AND T0101  ; 扫码位无料感应
AND T1383  ; 扫码阻挡气缸伸出延时
OR 1230.02  ; 扫码阻挡伸出
ANDLD
ANDNOT T0209  ; 扫码阻挡气缸伸出
OUT 1230.02  ; 扫码阻挡伸出

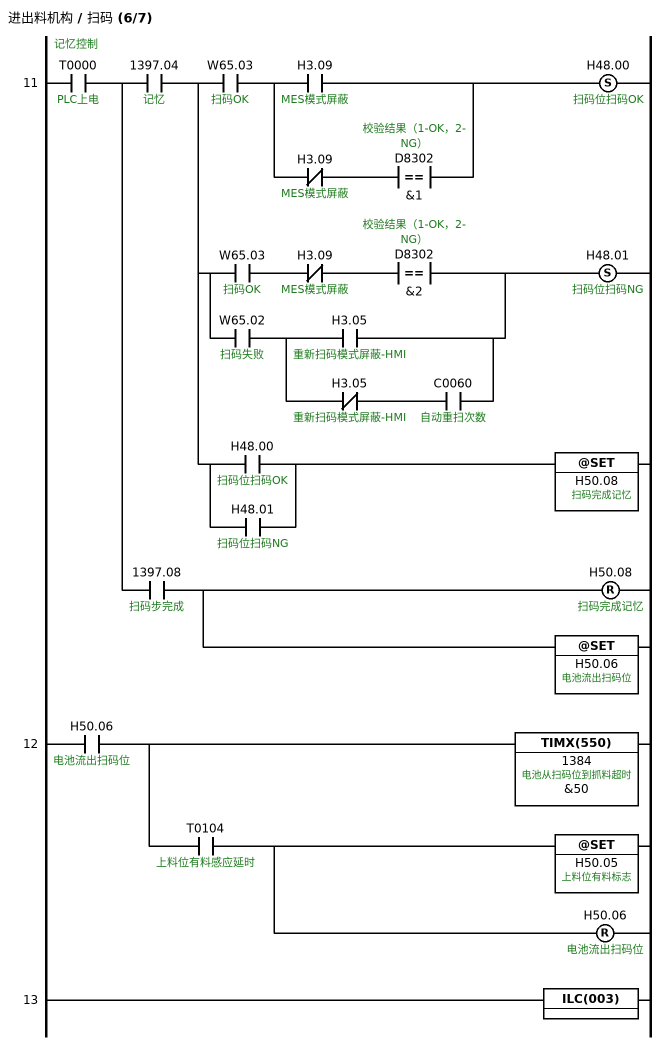
; rung 11: 记忆控制
LD T0000  ; PLC上电
OUT TR0
AND 1397.04  ; 记忆
OUT TR1
AND W65.03  ; 扫码OK
LD H3.09  ; MES模式屏蔽
LDNOT H3.09  ; MES模式屏蔽
AND=(300) D8302 &1  ; 校验结果（1-OK，2-NG）
ORLD
ANDLD
SET H48.00  ; 扫码位扫码OK
LD TR1
LD W65.03  ; 扫码OK
ANDNOT H3.09  ; MES模式屏蔽
AND=(300) D8302 &2  ; 校验结果（1-OK，2-NG）
LD W65.02  ; 扫码失败
LD H3.05  ; 重新扫码模式屏蔽-HMI
LDNOT H3.05  ; 重新扫码模式屏蔽-HMI
AND C0060  ; 自动重扫次数
ORLD
ANDLD
ORLD
ANDLD
SET H48.01  ; 扫码位扫码NG
LD TR1
LD H48.00  ; 扫码位扫码OK
OR H48.01  ; 扫码位扫码NG
ANDLD
@SET H50.08  ; 扫码完成记忆
LD TR0
AND 1397.08  ; 扫码步完成
RSET H50.08  ; 扫码完成记忆
@SET H50.06  ; 电池流出扫码位
; rung 12
LD H50.06  ; 电池流出扫码位
TIMX(550) 1384 &50  ; 电池从扫码位到抓料超时
AND T0104  ; 上料位有料感应延时
@SET H50.05  ; 上料位有料标志
RSET H50.06  ; 电池流出扫码位
; rung 13
ILC(003)

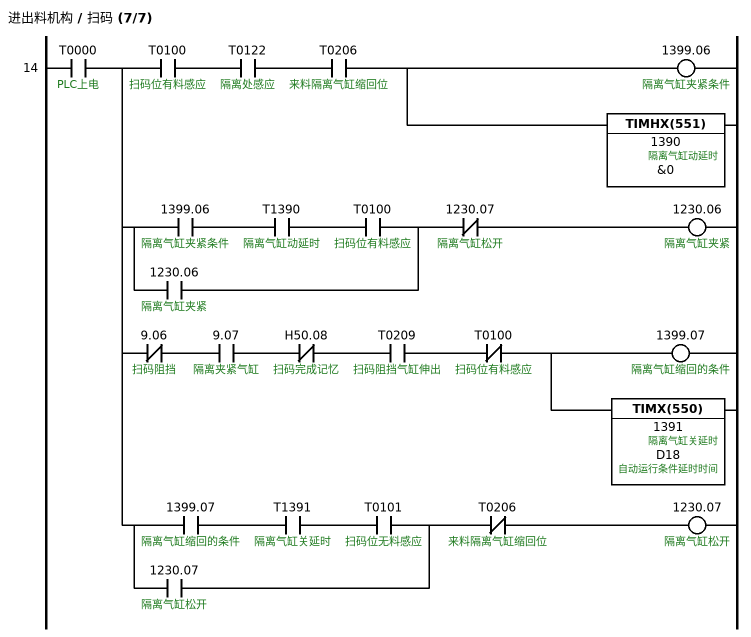
; rung 14
LD T0000  ; PLC上电
OUT TR0
AND T0100  ; 扫码位有料感应
AND T0122  ; 隔离处感应
AND T0206  ; 来料隔离气缸缩回位
OUT 1399.06  ; 隔离气缸夹紧条件
TIMHX(551) 1390 &0  ; 隔离气缸动延时
LD TR0
LD 1399.06  ; 隔离气缸夹紧条件
AND T1390  ; 隔离气缸动延时
AND T0100  ; 扫码位有料感应
OR 1230.06  ; 隔离气缸夹紧
ANDLD
ANDNOT 1230.07  ; 隔离气缸松开
OUT 1230.06  ; 隔离气缸夹紧
LD TR0
ANDNOT 9.06  ; 扫码阻挡
AND 9.07  ; 隔离夹紧气缸
ANDNOT H50.08  ; 扫码完成记忆
AND T0209  ; 扫码阻挡气缸伸出
ANDNOT T0100  ; 扫码位有料感应
OUT 1399.07  ; 隔离气缸缩回的条件
TIMX(550) 1391 D18  ; 自动运行条件延时时间, 隔离气缸关延时
LD TR0
LD 1399.07  ; 隔离气缸缩回的条件
AND T1391  ; 隔离气缸关延时
AND T0101  ; 扫码位无料感应
OR 1230.07  ; 隔离气缸松开
ANDLD
ANDNOT T0206  ; 来料隔离气缸缩回位
OUT 1230.07  ; 隔离气缸松开

### Section 进料手动

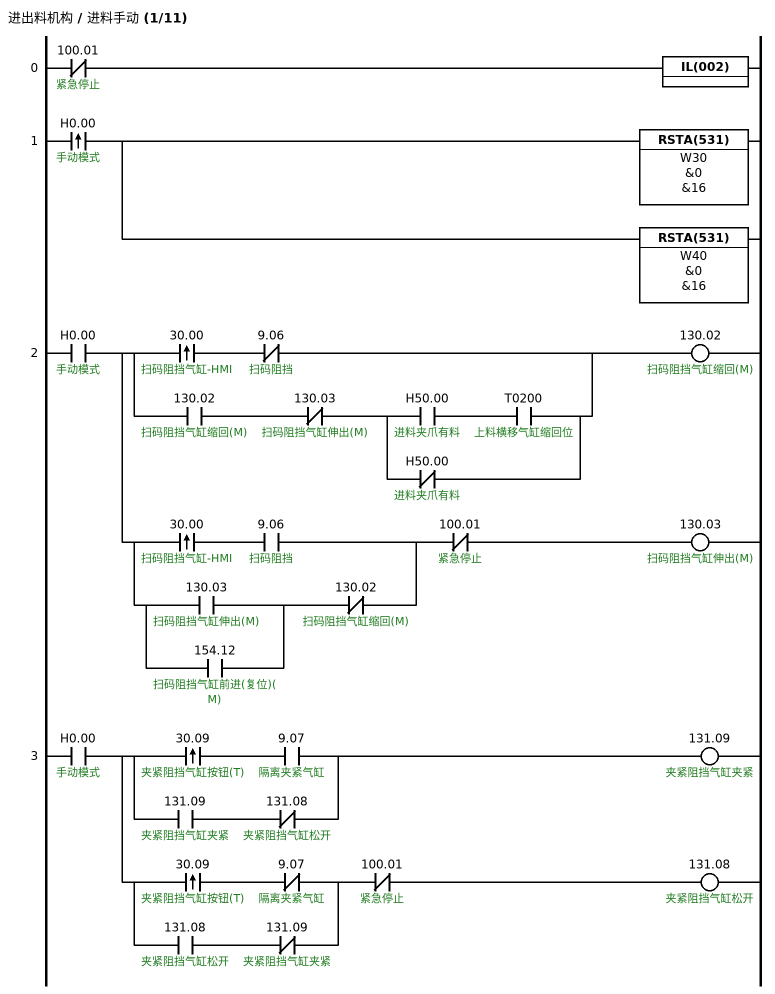
; rung 0
LDNOT 100.01  ; 紧急停止
IL(002)
; rung 1
@LD H0.00  ; 手动模式
RSTA(531) W30 &0 &16
RSTA(531) W40 &0 &16
; rung 2
LD H0.00  ; 手动模式
OUT TR0
@LD 30.00  ; 扫码阻挡气缸-HMI
ANDNOT 9.06  ; 扫码阻挡
LD 130.02  ; 扫码阻挡气缸缩回(M)
ANDNOT 130.03  ; 扫码阻挡气缸伸出(M)
LD H50.00  ; 进料夹爪有料
AND T0200  ; 上料横移气缸缩回位
ORNOT H50.00  ; 进料夹爪有料
ANDLD
ORLD
ANDLD
OUT 130.02  ; 扫码阻挡气缸缩回(M)
LD TR0
@LD 30.00  ; 扫码阻挡气缸-HMI
AND 9.06  ; 扫码阻挡
LD 130.03  ; 扫码阻挡气缸伸出(M)
OR 154.12  ; 扫码阻挡气缸前进(复位)(M)
ANDNOT 130.02  ; 扫码阻挡气缸缩回(M)
ORLD
ANDLD
ANDNOT 100.01  ; 紧急停止
OUT 130.03  ; 扫码阻挡气缸伸出(M)
; rung 3
LD H0.00  ; 手动模式
OUT TR0
@LD 30.09  ; 夹紧阻挡气缸按钮(T)
AND 9.07  ; 隔离夹紧气缸
LD 131.09  ; 夹紧阻挡气缸夹紧
ANDNOT 131.08  ; 夹紧阻挡气缸松开
ORLD
ANDLD
OUT 131.09  ; 夹紧阻挡气缸夹紧
LD TR0
@LD 30.09  ; 夹紧阻挡气缸按钮(T)
ANDNOT 9.07  ; 隔离夹紧气缸
LD 131.08  ; 夹紧阻挡气缸松开
ANDNOT 131.09  ; 夹紧阻挡气缸夹紧
ORLD
ANDLD
ANDNOT 100.01  ; 紧急停止
OUT 131.08  ; 夹紧阻挡气缸松开

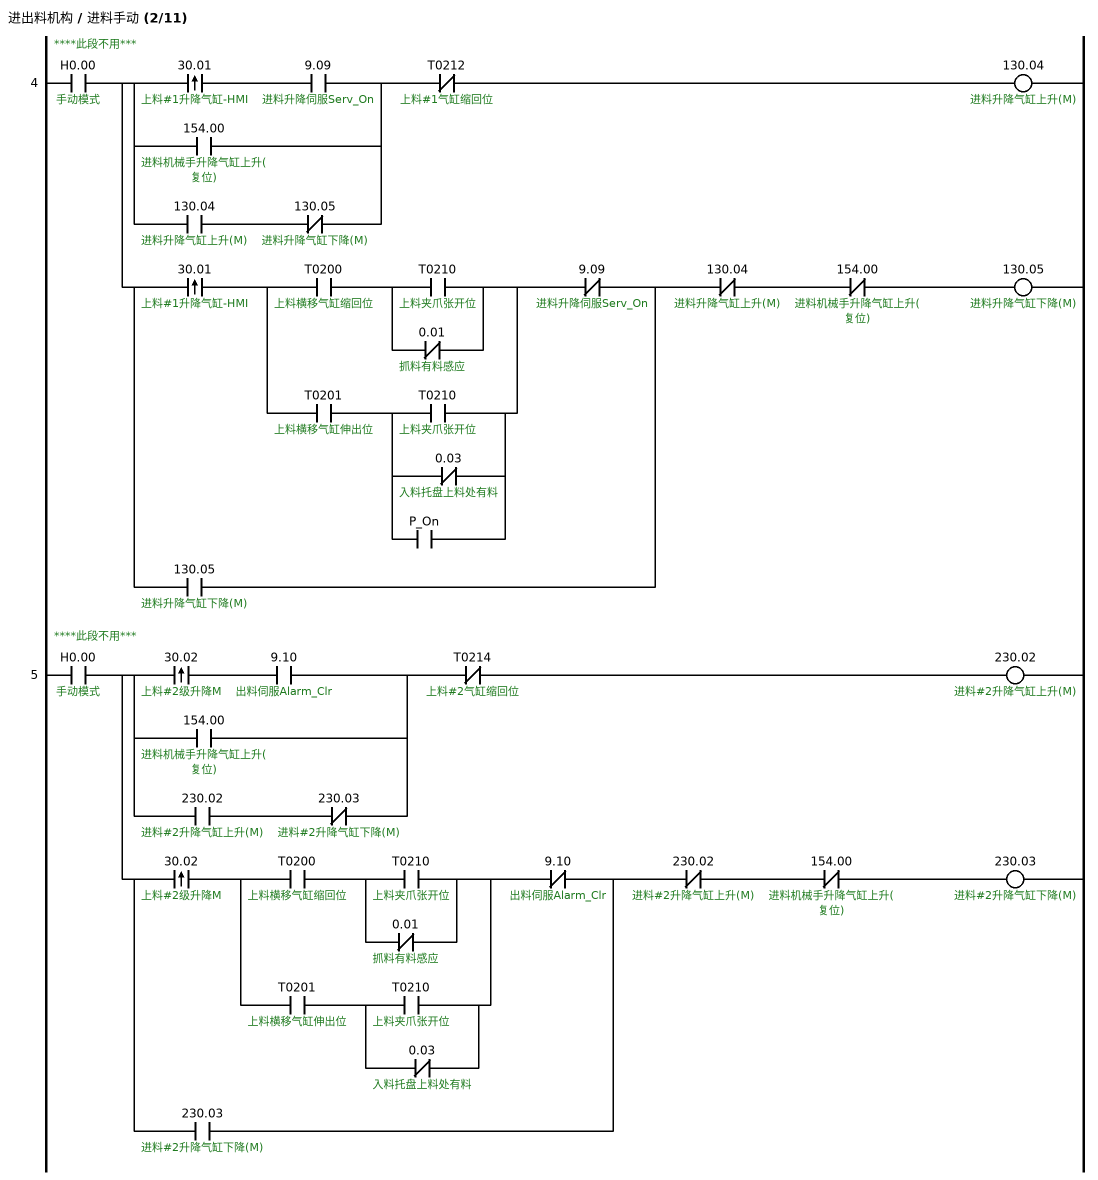
; rung 4: ****此段不用***
LD H0.00  ; 手动模式
OUT TR0
@LD 30.01  ; 上料#1升降气缸-HMI
AND 9.09  ; 进料升降伺服Serv_On
OR 154.00  ; 进料机械手升降气缸上升(复位)
LD 130.04  ; 进料升降气缸上升(M)
ANDNOT 130.05  ; 进料升降气缸下降(M)
ORLD
ANDLD
ANDNOT T0212  ; 上料#1气缸缩回位
OUT 130.04  ; 进料升降气缸上升(M)
LD TR0
@LD 30.01  ; 上料#1升降气缸-HMI
LD T0200  ; 上料横移气缸缩回位
LD T0210  ; 上料夹爪张开位
ORNOT 0.01  ; 抓料有料感应
ANDLD
LD T0201  ; 上料横移气缸伸出位
LD T0210  ; 上料夹爪张开位
ORNOT 0.03  ; 入料托盘上料处有料
OR P_On
ANDLD
ORLD
ANDLD
ANDNOT 9.09  ; 进料升降伺服Serv_On
OR 130.05  ; 进料升降气缸下降(M)
ANDLD
ANDNOT 130.04  ; 进料升降气缸上升(M)
ANDNOT 154.00  ; 进料机械手升降气缸上升(复位)
OUT 130.05  ; 进料升降气缸下降(M)
; rung 5: ****此段不用***
LD H0.00  ; 手动模式
OUT TR0
@LD 30.02  ; 上料#2级升降M
AND 9.10  ; 出料伺服Alarm_Clr
OR 154.00  ; 进料机械手升降气缸上升(复位)
LD 230.02  ; 进料#2升降气缸上升(M)
ANDNOT 230.03  ; 进料#2升降气缸下降(M)
ORLD
ANDLD
ANDNOT T0214  ; 上料#2气缸缩回位
OUT 230.02  ; 进料#2升降气缸上升(M)
LD TR0
@LD 30.02  ; 上料#2级升降M
LD T0200  ; 上料横移气缸缩回位
LD T0210  ; 上料夹爪张开位
ORNOT 0.01  ; 抓料有料感应
ANDLD
LD T0201  ; 上料横移气缸伸出位
LD T0210  ; 上料夹爪张开位
ORNOT 0.03  ; 入料托盘上料处有料
ANDLD
ORLD
ANDLD
ANDNOT 9.10  ; 出料伺服Alarm_Clr
OR 230.03  ; 进料#2升降气缸下降(M)
ANDLD
ANDNOT 230.02  ; 进料#2升降气缸上升(M)
ANDNOT 154.00  ; 进料机械手升降气缸上升(复位)
OUT 230.03  ; 进料#2升降气缸下降(M)

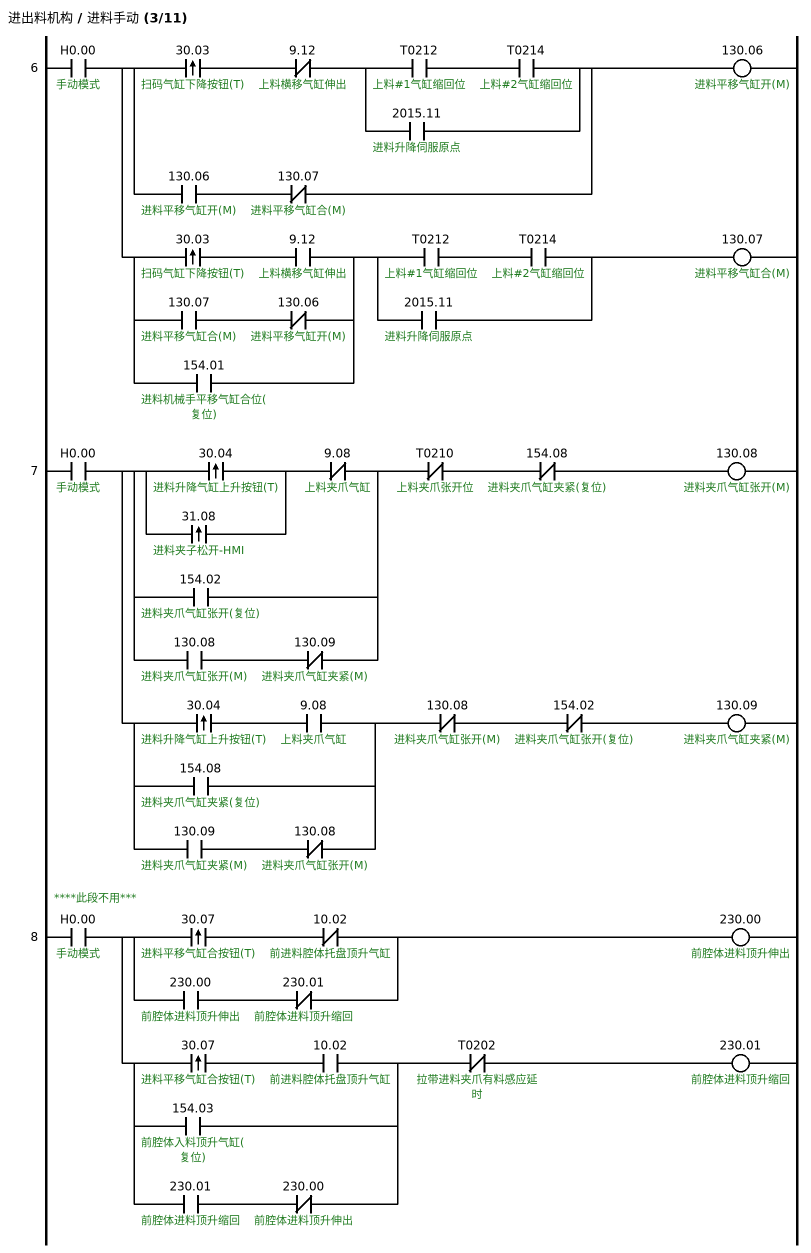
; rung 6
LD H0.00  ; 手动模式
OUT TR0
@LD 30.03  ; 扫码气缸下降按钮(T)
ANDNOT 9.12  ; 上料横移气缸伸出
LD T0212  ; 上料#1气缸缩回位
AND T0214  ; 上料#2气缸缩回位
OR 2015.11  ; 进料升降伺服原点
ANDLD
LD 130.06  ; 进料平移气缸开(M)
ANDNOT 130.07  ; 进料平移气缸合(M)
ORLD
ANDLD
OUT 130.06  ; 进料平移气缸开(M)
LD TR0
@LD 30.03  ; 扫码气缸下降按钮(T)
AND 9.12  ; 上料横移气缸伸出
LD 130.07  ; 进料平移气缸合(M)
ANDNOT 130.06  ; 进料平移气缸开(M)
ORLD
OR 154.01  ; 进料机械手平移气缸合位(复位)
ANDLD
LD T0212  ; 上料#1气缸缩回位
AND T0214  ; 上料#2气缸缩回位
OR 2015.11  ; 进料升降伺服原点
ANDLD
OUT 130.07  ; 进料平移气缸合(M)
; rung 7
LD H0.00  ; 手动模式
OUT TR0
@LD 30.04  ; 进料升降气缸上升按钮(T)
@OR 31.08  ; 进料夹子松开-HMI
ANDNOT 9.08  ; 上料夹爪气缸
OR 154.02  ; 进料夹爪气缸张开(复位)
LD 130.08  ; 进料夹爪气缸张开(M)
ANDNOT 130.09  ; 进料夹爪气缸夹紧(M)
ORLD
ANDLD
ANDNOT T0210  ; 上料夹爪张开位
ANDNOT 154.08  ; 进料夹爪气缸夹紧(复位)
OUT 130.08  ; 进料夹爪气缸张开(M)
LD TR0
@LD 30.04  ; 进料升降气缸上升按钮(T)
AND 9.08  ; 上料夹爪气缸
OR 154.08  ; 进料夹爪气缸夹紧(复位)
LD 130.09  ; 进料夹爪气缸夹紧(M)
ANDNOT 130.08  ; 进料夹爪气缸张开(M)
ORLD
ANDLD
ANDNOT 130.08  ; 进料夹爪气缸张开(M)
ANDNOT 154.02  ; 进料夹爪气缸张开(复位)
OUT 130.09  ; 进料夹爪气缸夹紧(M)
; rung 8: ****此段不用***
LD H0.00  ; 手动模式
OUT TR0
@LD 30.07  ; 进料平移气缸合按钮(T)
ANDNOT 10.02  ; 前进料腔体托盘顶升气缸
LD 230.00  ; 前腔体进料顶升伸出
ANDNOT 230.01  ; 前腔体进料顶升缩回
ORLD
ANDLD
OUT 230.00  ; 前腔体进料顶升伸出
LD TR0
@LD 30.07  ; 进料平移气缸合按钮(T)
AND 10.02  ; 前进料腔体托盘顶升气缸
OR 154.03  ; 前腔体入料顶升气缸(复位)
LD 230.01  ; 前腔体进料顶升缩回
ANDNOT 230.00  ; 前腔体进料顶升伸出
ORLD
ANDLD
ANDNOT T0202  ; 拉带进料夹爪有料感应延时
OUT 230.01  ; 前腔体进料顶升缩回

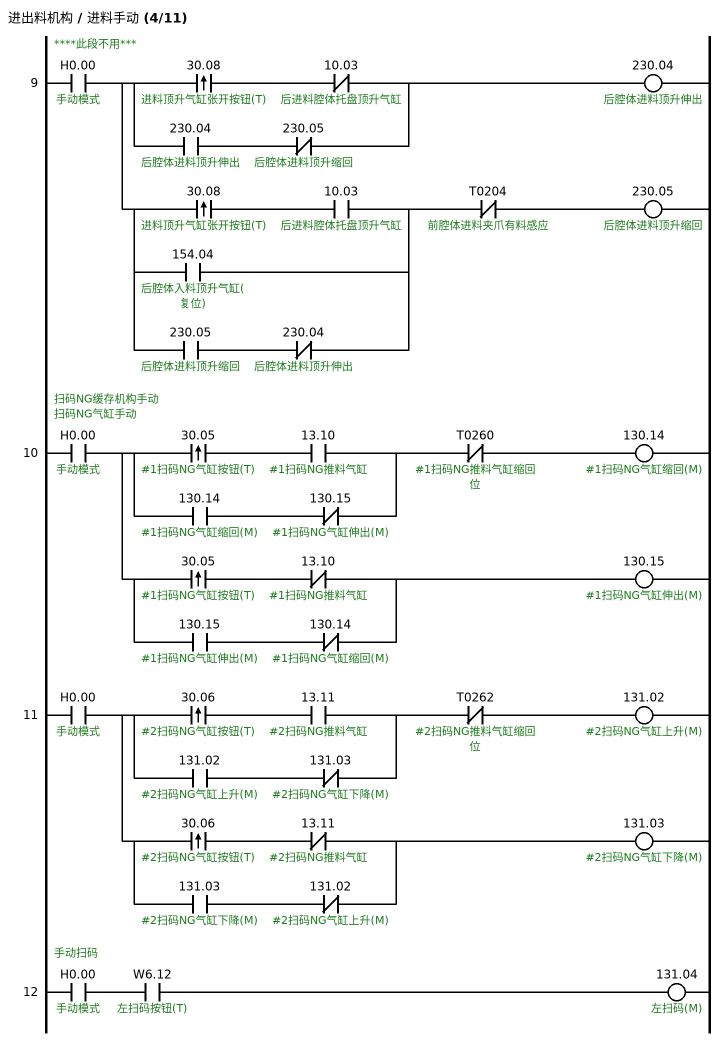
; rung 9: ****此段不用***
LD H0.00  ; 手动模式
OUT TR0
@LD 30.08  ; 进料顶升气缸张开按钮(T)
ANDNOT 10.03  ; 后进料腔体托盘顶升气缸
LD 230.04  ; 后腔体进料顶升伸出
ANDNOT 230.05  ; 后腔体进料顶升缩回
ORLD
ANDLD
OUT 230.04  ; 后腔体进料顶升伸出
LD TR0
@LD 30.08  ; 进料顶升气缸张开按钮(T)
AND 10.03  ; 后进料腔体托盘顶升气缸
OR 154.04  ; 后腔体入料顶升气缸(复位)
LD 230.05  ; 后腔体进料顶升缩回
ANDNOT 230.04  ; 后腔体进料顶升伸出
ORLD
ANDLD
ANDNOT T0204  ; 前腔体进料夹爪有料感应
OUT 230.05  ; 后腔体进料顶升缩回
; rung 10: 扫码NG缓存机构手动 / 扫码NG气缸手动
LD H0.00  ; 手动模式
OUT TR0
@LD 30.05  ; #1扫码NG气缸按钮(T)
AND 13.10  ; #1扫码NG推料气缸
LD 130.14  ; #1扫码NG气缸缩回(M)
ANDNOT 130.15  ; #1扫码NG气缸伸出(M)
ORLD
ANDLD
ANDNOT T0260  ; #1扫码NG推料气缸缩回位
OUT 130.14  ; #1扫码NG气缸缩回(M)
LD TR0
@LD 30.05  ; #1扫码NG气缸按钮(T)
ANDNOT 13.10  ; #1扫码NG推料气缸
LD 130.15  ; #1扫码NG气缸伸出(M)
ANDNOT 130.14  ; #1扫码NG气缸缩回(M)
ORLD
ANDLD
OUT 130.15  ; #1扫码NG气缸伸出(M)
; rung 11
LD H0.00  ; 手动模式
OUT TR0
@LD 30.06  ; #2扫码NG气缸按钮(T)
AND 13.11  ; #2扫码NG推料气缸
LD 131.02  ; #2扫码NG气缸上升(M)
ANDNOT 131.03  ; #2扫码NG气缸下降(M)
ORLD
ANDLD
ANDNOT T0262  ; #2扫码NG推料气缸缩回位
OUT 131.02  ; #2扫码NG气缸上升(M)
LD TR0
@LD 30.06  ; #2扫码NG气缸按钮(T)
ANDNOT 13.11  ; #2扫码NG推料气缸
LD 131.03  ; #2扫码NG气缸下降(M)
ANDNOT 131.02  ; #2扫码NG气缸上升(M)
ORLD
ANDLD
OUT 131.03  ; #2扫码NG气缸下降(M)
; rung 12: 手动扫码
LD H0.00  ; 手动模式
AND W6.12  ; 左扫码按钮(T)
OUT 131.04  ; 左扫码(M)

